LIN {X 0,Y 367.109,Z 392.803,A -85,B 0,C 180,E1 -12833.598,E2 -12833.598} C_VEL
LIN {X 0,Y 367.142,Z 392.339,A -85,B 0,C 180,E1 -12835.398,E2 -12835.398} C_VEL
LIN {X 0,Y 367.242,Z 390.593,A -85,B 0,C 180,E1 -12837.355,E2 -12837.355} C_VEL
LIN {X 0,Y 367.556,Z 387.382,A -85,B 0,C 180,E1 -12839.365,E2 -12839.365} C_VEL
LIN {X 0,Y 367.902,Z 382.367,A -85,B 0,C 180,E1 -12841.489,E2 -12841.489} C_VEL
LIN {X 0,Y 368.375,Z 376.663,A -85,B 0,C 180,E1 -12843.259,E2 -12843.259} C_VEL
LIN {X 0,Y 368.98,Z 369.858,A -85,B 0,C 180,E1 -12844.927,E2 -12844.927} C_VEL
LIN {X 0,Y 369.688,Z 362.048,A -85,B 0,C 180,E1 -12846.472,E2 -12846.472} C_VEL
LIN {X 0,Y 370.635,Z 352.269,A -85,B 0,C 180,E1 -12848.024,E2 -12848.024} C_VEL
LIN {X 0,Y 371.602,Z 341.593,A -85,B 0,C 180,E1 -12849.377,E2 -12849.377} C_VEL
LIN {X 0,Y 372.49,Z 331.477,A -85,B 0,C 180,E1 -12850.406,E2 -12850.406} C_VEL
LIN {X 0,Y 373.295,Z 320.016,A -85,B 0,C 180,E1 -12851.335,E2 -12851.335} C_VEL
LIN {X 0,Y 373.997,Z 307.877,A -85,B 0,C 180,E1 -12852.08,E2 -12852.08} C_VEL
LIN {X 0,Y 374.667,Z 294.33,A -85,B 0,C 180,E1 -12852.665,E2 -12852.665} C_VEL
LIN {X 0,Y 375.041,Z 279.803,A -85,B 0,C 180,E1 -12853.034,E2 -12853.034} C_VEL
LIN {X 0,Y 376.225,Z 207.722,A -85,B 0,C 180,E1 -12854.477,E2 -12854.477} C_VEL
LIN {X 0,Y 371.538,Z 182.162,A -85,B 0,C 180,E1 -12855.285,E2 -12855.285} C_VEL
LIN {X 0,Y 371.499,Z 181.295,A -85,B 0,C 180,E1 -12855.398,E2 -12855.398} C_VEL
LIN {X 0,Y 371.537,Z 177.576,A -85,B 0,C 180,E1 -12856.324,E2 -12856.324} C_VEL
LIN {X 0,Y 369.73,Z 167.61,A -85,B 0,C 180,E1 -12859.044,E2 -12859.044} C_VEL
LIN {X 0,Y 369.072,Z 164.061,A -85,B 0,C 180,E1 -12860.099,E2 -12860.099} C_VEL
LIN {X 0,Y 369.199,Z 163.994,A -85,B 0,C 180,E1 -12863.443,E2 -12863.443} C_VEL
LIN {X 0,Y 369.313,Z 163.984,A -85,B 0,C 180,E1 -12867.82,E2 -12867.82} C_VEL
LIN {X 0,Y 369.454,Z 163.964,A -85,B 0,C 180,E1 -12870.001,E2 -12870.001} C_VEL
LIN {X 0,Y 369.314,Z 163.98,A -85,B 0,C 180,E1 -12872.182,E2 -12872.182} C_VEL
LIN {X 0,Y 369.049,Z 164.011,A -85,B 0,C 180,E1 -12873.745,E2 -12873.745} C_VEL
LIN {X 0,Y 368.326,Z 164.102,A -85,B 0,C 180,E1 -12874.657,E2 -12874.657} C_VEL
LIN {X 0,Y 365.524,Z 164.452,A -85,B 0,C 180,E1 -12876.141,E2 -12876.141} C_VEL
LIN {X 0,Y 363.181,Z 164.746,A -85,B 0,C 180,E1 -12877.342,E2 -12877.342} C_VEL
LIN {X 0,Y 362.157,Z 164.871,A -85,B 0,C 180,E1 -12878.269,E2 -12878.269} C_VEL
LIN {X 0,Y 362.061,Z 164.882,A -85,B 0,C 180,E1 -12878.583,E2 -12878.583} C_VEL
LIN {X 0,Y 361.959,Z 164.894,A -85,B 0,C 180,E1 -12882.333,E2 -12882.333} C_VEL
LIN {X 0,Y 361.961,Z 164.894,A -85,B 0,C 180,E1 -12884.621,E2 -12884.621} C_VEL
LIN {X 0,Y 361.955,Z 164.895,A -85,B 0,C 180,E1 -12888.1,E2 -12888.1} C_VEL
LIN {X 0,Y 361.891,Z 164.905,A -85,B 0,C 180,E1 -12891.654,E2 -12891.654} C_VEL
LIN {X 0,Y 361.927,Z 164.904,A -85,B 0,C 180,E1 -12895.291,E2 -12895.291} C_VEL
LIN {X 0,Y 361.908,Z 164.902,A -85,B 0,C 180,E1 -12897.78,E2 -12897.78} C_VEL
LIN {X 0,Y 361.837,Z 164.911,A -85,B 0,C 180,E1 -12901.63,E2 -12901.63} C_VEL
LIN {X 0,Y 361.874,Z 164.908,A -85,B 0,C 180,E1 -12905.346,E2 -12905.346} C_VEL
LIN {X 0,Y 361.868,Z 164.911,A -85,B 0,C 180,E1 -12909.027,E2 -12909.027} C_VEL
LIN {X 0,Y 361.836,Z 164.916,A -85,B 0,C 180,E1 -12912.83,E2 -12912.83} C_VEL
LIN {X 0,Y 361.819,Z 164.912,A -85,B 0,C 180,E1 -12915.947,E2 -12915.947} C_VEL
LIN {X 0,Y 361.83,Z 164.912,A -85,B 0,C 180,E1 -12919.246,E2 -12919.246} C_VEL
LIN {X 0,Y 361.864,Z 164.909,A -85,B 0,C 180,E1 -12922.982,E2 -12922.982} C_VEL
LIN {X 0,Y 361.859,Z 164.912,A -85,B 0,C 180,E1 -12926.631,E2 -12926.631} C_VEL
LIN {X 0,Y 361.857,Z 164.907,A -85,B 0,C 180,E1 -12929.671,E2 -12929.671} C_VEL
LIN {X 0,Y 361.873,Z 164.905,A -85,B 0,C 180,E1 -12933.469,E2 -12933.469} C_VEL
LIN {X 0,Y 361.883,Z 164.904,A -85,B 0,C 180,E1 -12937.145,E2 -12937.145} C_VEL
LIN {X 0,Y 361.907,Z 164.902,A -85,B 0,C 180,E1 -12940.724,E2 -12940.724} C_VEL
LIN {X 0,Y 361.933,Z 164.898,A -85,B 0,C 180,E1 -12943.067,E2 -12943.067} C_VEL
LIN {X 0,Y 362,Z 164.891,A -85,B 0,C 180,E1 -12946.528,E2 -12946.528} C_VEL
LIN {X 0,Y 362,Z 164.895,A -85,B 0,C 180,E1 -12949.938,E2 -12949.938} C_VEL
LIN {X 0,Y 362.122,Z 164.875,A -85,B 0,C 180,E1 -12953.313,E2 -12953.313} C_VEL
LIN {X 0,Y 362.265,Z 164.862,A -85,B 0,C 180,E1 -12957.777,E2 -12957.777} C_VEL
LIN {X 0,Y 362.269,Z 164.857,A -85,B 0,C 180,E1 -12962.224,E2 -12962.224} C_VEL
LIN {X 0,Y 362.117,Z 164.875,A -85,B 0,C 180,E1 -12966.688,E2 -12966.688} C_VEL
LIN {X 0,Y 361.999,Z 164.891,A -85,B 0,C 180,E1 -12970.063,E2 -12970.063} C_VEL
LIN {X 0,Y 362.001,Z 164.891,A -85,B 0,C 180,E1 -12973.899,E2 -12973.899} C_VEL
LIN {X 0,Y 361.929,Z 164.9,A -85,B 0,C 180,E1 -12976.935,E2 -12976.935} C_VEL
LIN {X 0,Y 361.878,Z 164.904,A -85,B 0,C 180,E1 -12980.462,E2 -12980.462} C_VEL
LIN {X 0,Y 361.864,Z 164.906,A -85,B 0,C 180,E1 -12984.101,E2 -12984.101} C_VEL
LIN {X 0,Y 361.836,Z 164.911,A -85,B 0,C 180,E1 -12987.786,E2 -12987.786} C_VEL
LIN {X 0,Y 361.829,Z 164.915,A -85,B 0,C 180,E1 -12991.28,E2 -12991.28} C_VEL
LIN {X 0,Y 361.853,Z 164.908,A -85,B 0,C 180,E1 -12994.281,E2 -12994.281} C_VEL
LIN {X 0,Y 361.859,Z 164.91,A -85,B 0,C 180,E1 -12997.221,E2 -12997.221} C_VEL
LIN {X 0,Y 361.813,Z 164.917,A -85,B 0,C 180,E1 -13000.751,E2 -13000.751} C_VEL
LIN {X 0,Y 361.814,Z 164.914,A -85,B 0,C 180,E1 -13004.37,E2 -13004.37} C_VEL
LIN {X 0,Y 361.825,Z 164.911,A -85,B 0,C 180,E1 -13007.571,E2 -13007.571} C_VEL
LIN {X 0,Y 361.842,Z 164.909,A -85,B 0,C 180,E1 -13011.571,E2 -13011.571} C_VEL
LIN {X 0,Y 361.865,Z 164.912,A -85,B 0,C 180,E1 -13014.658,E2 -13014.658} C_VEL
LIN {X 0,Y 361.822,Z 164.916,A -85,B 0,C 180,E1 -13018.368,E2 -13018.368} C_VEL
LIN {X 0,Y 361.909,Z 165.145,A -85,B 0,C 180,E1 -13021.392,E2 -13021.392} C_VEL
LIN {X 0,Y 364.539,Z 178.239,A -85,B 0,C 180,E1 -13024.903,E2 -13024.903} C_VEL
LIN {X 0,Y 365.265,Z 183.174,A -85,B 0,C 180,E1 -13026.167,E2 -13026.167} C_VEL
LIN {X 0,Y 364.446,Z 192.349,A -85,B 0,C 180,E1 -13028.323,E2 -13028.323} C_VEL
LIN {X 0,Y 365.484,Z 198.9,A -85,B 0,C 180,E1 -13028.57,E2 -13028.57} C_VEL
LIN {X 0,Y 369.443,Z 223.822,A -85,B 0,C 180,E1 -13029.318,E2 -13029.318} C_VEL
LIN {X 0,Y 367.995,Z 300.62,A -85,B 0,C 180,E1 -13030.909,E2 -13030.909} C_VEL
LIN {X 0,Y 367.351,Z 314.312,A -85,B 0,C 180,E1 -13031.417,E2 -13031.417} C_VEL
LIN {X 0,Y 366.485,Z 327.23,A -85,B 0,C 180,E1 -13032.131,E2 -13032.131} C_VEL
LIN {X 0,Y 365.522,Z 339.819,A -85,B 0,C 180,E1 -13033.092,E2 -13033.092} C_VEL
LIN {X 0,Y 364.556,Z 351.066,A -85,B 0,C 180,E1 -13034.198,E2 -13034.198} C_VEL
LIN {X 0,Y 363.668,Z 361.183,A -85,B 0,C 180,E1 -13035.449,E2 -13035.449} C_VEL
LIN {X 0,Y 362.79,Z 370.328,A -85,B 0,C 180,E1 -13036.842,E2 -13036.842} C_VEL
LIN {X 0,Y 361.84,Z 379.24,A -85,B 0,C 180,E1 -13038.516,E2 -13038.516} C_VEL
LIN {X 0,Y 361.199,Z 386.366,A -85,B 0,C 180,E1 -13040.196,E2 -13040.196} C_VEL
LIN {X 0,Y 360.687,Z 392.862,A -85,B 0,C 180,E1 -13042.16,E2 -13042.16} C_VEL
LIN {X 0,Y 360.428,Z 397.403,A -85,B 0,C 180,E1 -13043.965,E2 -13043.965} C_VEL
LIN {X 0,Y 360.348,Z 400.313,A -85,B 0,C 180,E1 -13045.525,E2 -13045.525} C_VEL
LIN {X 0,Y 360.275,Z 401.892,A -85,B 0,C 180,E1 -13046.644,E2 -13046.644} C_VEL
LIN {X 0,Y 360.226,Z 403.034,A -85,B 0,C 180,E1 -13047.763,E2 -13047.763} C_VEL
LIN {X 0,Y 360.252,Z 403.744,A -85,B 0,C 180,E1 -13048.881,E2 -13048.881} C_VEL
LIN {X 0,Y 360.291,Z 404.061,A -85,B 0,C 180,E1 -13049.999,E2 -13049.999} C_VEL
LIN {X 0,Y 360.25,Z 403.987,A -85,B 0,C 180,E1 -13051.117,E2 -13051.117} C_VEL
LIN {X 0,Y 360.225,Z 403.495,A -85,B 0,C 180,E1 -13052.235,E2 -13052.235} C_VEL
LIN {X 0,Y 360.278,Z 402.578,A -85,B 0,C 180,E1 -13053.354,E2 -13053.354} C_VEL
LIN {X 0,Y 360.379,Z 401.262,A -85,B 0,C 180,E1 -13054.473,E2 -13054.473} C_VEL
LIN {X 0,Y 360.463,Z 398.611,A -85,B 0,C 180,E1 -13056.087,E2 -13056.087} C_VEL
LIN {X 0,Y 360.756,Z 394.67,A -85,B 0,C 180,E1 -13057.836,E2 -13057.836} C_VEL
LIN {X 0,Y 361.219,Z 389.732,A -85,B 0,C 180,E1 -13059.518,E2 -13059.518} C_VEL
LIN {X 0,Y 361.871,Z 383.528,A -85,B 0,C 180,E1 -13061.197,E2 -13061.197} C_VEL
LIN {X 0,Y 362.818,Z 375.82,A -85,B 0,C 180,E1 -13062.87,E2 -13062.87} C_VEL
LIN {X 0,Y 364.016,Z 366.15,A -85,B 0,C 180,E1 -13064.535,E2 -13064.535} C_VEL
LIN {X 0,Y 365.018,Z 356.196,A -85,B 0,C 180,E1 -13065.923,E2 -13065.923} C_VEL
LIN {X 0,Y 366.289,Z 344.984,A -85,B 0,C 180,E1 -13067.156,E2 -13067.156} C_VEL
LIN {X 0,Y 367.386,Z 334.036,A -85,B 0,C 180,E1 -13068.109,E2 -13068.109} C_VEL
LIN {X 0,Y 368.435,Z 321.974,A -85,B 0,C 180,E1 -13068.92,E2 -13068.92} C_VEL
LIN {X 0,Y 369.204,Z 309.573,A -85,B 0,C 180,E1 -13069.529,E2 -13069.529} C_VEL
LIN {X 0,Y 369.741,Z 295.528,A -85,B 0,C 180,E1 -13069.97,E2 -13069.97} C_VEL
LIN {X 0,Y 371.27,Z 223.76,A -85,B 0,C 180,E1 -13071.458,E2 -13071.458} C_VEL
LIN {X 0,Y 367.556,Z 202.377,A -85,B 0,C 180,E1 -13072.204,E2 -13072.204} C_VEL
LIN {X 0,Y 365.353,Z 191.898,A -85,B 0,C 180,E1 -13072.644,E2 -13072.644} C_VEL
LIN {X 0,Y 365.684,Z 187.966,A -85,B 0,C 180,E1 -13073.501,E2 -13073.501} C_VEL
LIN {X 0,Y 365.843,Z 184.32,A -85,B 0,C 180,E1 -13074.393,E2 -13074.393} C_VEL
LIN {X 0,Y 364.208,Z 175.338,A -85,B 0,C 180,E1 -13076.802,E2 -13076.802} C_VEL
LIN {X 0,Y 361.879,Z 164.958,A -85,B 0,C 180,E1 -13079.803,E2 -13079.803} C_VEL
LIN {X 0,Y 361.853,Z 164.907,A -85,B 0,C 180,E1 -13083.367,E2 -13083.367} C_VEL
LIN {X 0,Y 361.855,Z 164.911,A -85,B 0,C 180,E1 -13087.017,E2 -13087.017} C_VEL
LIN {X 0,Y 361.804,Z 164.917,A -85,B 0,C 180,E1 -13090.749,E2 -13090.749} C_VEL
LIN {X 0,Y 361.804,Z 164.914,A -85,B 0,C 180,E1 -13094.368,E2 -13094.368} C_VEL
LIN {X 0,Y 361.814,Z 164.918,A -85,B 0,C 180,E1 -13097.569,E2 -13097.569} C_VEL
LIN {X 0,Y 361.834,Z 164.91,A -85,B 0,C 180,E1 -13101.57,E2 -13101.57} C_VEL
LIN {X 0,Y 361.861,Z 164.91,A -85,B 0,C 180,E1 -13104.655,E2 -13104.655} C_VEL
LIN {X 0,Y 361.828,Z 164.912,A -85,B 0,C 180,E1 -13108.369,E2 -13108.369} C_VEL
LIN {X 0,Y 361.856,Z 164.913,A -85,B 0,C 180,E1 -13110.951,E2 -13110.951} C_VEL
LIN {X 0,Y 361.869,Z 164.91,A -85,B 0,C 180,E1 -13114.705,E2 -13114.705} C_VEL
LIN {X 0,Y 361.849,Z 164.909,A -85,B 0,C 180,E1 -13118.344,E2 -13118.344} C_VEL
LIN {X 0,Y 361.909,Z 164.9,A -85,B 0,C 180,E1 -13122.084,E2 -13122.084} C_VEL
LIN {X 0,Y 361.95,Z 164.894,A -85,B 0,C 180,E1 -13125.379,E2 -13125.379} C_VEL
LIN {X 0,Y 361.957,Z 164.892,A -85,B 0,C 180,E1 -13128.803,E2 -13128.803} C_VEL
LIN {X 0,Y 362.082,Z 164.879,A -85,B 0,C 180,E1 -13132.191,E2 -13132.191} C_VEL
LIN {X 0,Y 362.089,Z 164.881,A -85,B 0,C 180,E1 -13134.43,E2 -13134.43} C_VEL
LIN {X 0,Y 362.255,Z 164.858,A -85,B 0,C 180,E1 -13137.776,E2 -13137.776} C_VEL
LIN {X 0,Y 362.252,Z 164.863,A -85,B 0,C 180,E1 -13142.223,E2 -13142.223} C_VEL
LIN {X 0,Y 362.127,Z 164.875,A -85,B 0,C 180,E1 -13146.686,E2 -13146.686} C_VEL
LIN {X 0,Y 361.982,Z 164.894,A -85,B 0,C 180,E1 -13150.063,E2 -13150.063} C_VEL
LIN {X 0,Y 361.985,Z 164.893,A -85,B 0,C 180,E1 -13153.898,E2 -13153.898} C_VEL
LIN {X 0,Y 361.915,Z 164.904,A -85,B 0,C 180,E1 -13156.934,E2 -13156.934} C_VEL
LIN {X 0,Y 361.87,Z 164.91,A -85,B 0,C 180,E1 -13160.461,E2 -13160.461} C_VEL
LIN {X 0,Y 361.848,Z 164.915,A -85,B 0,C 180,E1 -13164.101,E2 -13164.101} C_VEL
LIN {X 0,Y 361.861,Z 165.115,A -85,B 0,C 180,E1 -13166.7,E2 -13166.7} C_VEL
LIN {X 0,Y 364.298,Z 175.702,A -85,B 0,C 180,E1 -13169.761,E2 -13169.761} C_VEL
LIN {X 0,Y 365.43,Z 181.869,A -85,B 0,C 180,E1 -13171.387,E2 -13171.387} C_VEL
LIN {X 0,Y 366.56,Z 185.876,A -85,B 0,C 180,E1 -13171.619,E2 -13171.619} C_VEL
LIN {X 0,Y 370.397,Z 203.475,A -85,B 0,C 180,E1 -13172.3,E2 -13172.3} C_VEL
LIN {X 0,Y 371.577,Z 210.184,A -85,B 0,C 180,E1 -13172.534,E2 -13172.534} C_VEL
LIN {X 0,Y 369.736,Z 290.324,A -85,B 0,C 180,E1 -13174.219,E2 -13174.219} C_VEL
LIN {X 0,Y 369.122,Z 303.569,A -85,B 0,C 180,E1 -13174.721,E2 -13174.721} C_VEL
LIN {X 0,Y 368.374,Z 315.12,A -85,B 0,C 180,E1 -13175.357,E2 -13175.357} C_VEL
LIN {X 0,Y 367.382,Z 327.182,A -85,B 0,C 180,E1 -13176.248,E2 -13176.248} C_VEL
LIN {X 0,Y 366.166,Z 339.44,A -85,B 0,C 180,E1 -13177.431,E2 -13177.431} C_VEL
LIN {X 0,Y 364.915,Z 350.146,A -85,B 0,C 180,E1 -13178.742,E2 -13178.742} C_VEL
LIN {X 0,Y 363.768,Z 359.977,A -85,B 0,C 180,E1 -13180.261,E2 -13180.261} C_VEL
LIN {X 0,Y 362.806,Z 367.927,A -85,B 0,C 180,E1 -13181.776,E2 -13181.776} C_VEL
LIN {X 0,Y 361.922,Z 374.835,A -85,B 0,C 180,E1 -13183.394,E2 -13183.394} C_VEL
LIN {X 0,Y 361.379,Z 380.255,A -85,B 0,C 180,E1 -13184.978,E2 -13184.978} C_VEL
LIN {X 0,Y 360.798,Z 385.639,A -85,B 0,C 180,E1 -13187.021,E2 -13187.021} C_VEL
LIN {X 0,Y 360.557,Z 388.562,A -85,B 0,C 180,E1 -13188.494,E2 -13188.494} C_VEL
LIN {X 0,Y 360.302,Z 390.657,A -85,B 0,C 180,E1 -13189.935,E2 -13189.935} C_VEL
LIN {X 0,Y 360.123,Z 392.042,A -85,B 0,C 180,E1 -13191.357,E2 -13191.357} C_VEL
LIN {X 0,Y 360.005,Z 392.863,A -85,B 0,C 180,E1 -13193.167,E2 -13193.167} C_VEL
LIN {X 0,Y 360.039,Z 392.591,A -85,B 0,C 180,E1 -13195.068,E2 -13195.068} C_VEL
LIN {X 0,Y 360.11,Z 391.067,A -85,B 0,C 180,E1 -13197.055,E2 -13197.055} C_VEL
LIN {X 0,Y 360.416,Z 388.143,A -85,B 0,C 180,E1 -13199.09,E2 -13199.09} C_VEL
LIN {X 0,Y 360.663,Z 384.41,A -85,B 0,C 180,E1 -13200.848,E2 -13200.848} C_VEL
LIN {X 0,Y 361.144,Z 378.85,A -85,B 0,C 180,E1 -13202.788,E2 -13202.788} C_VEL
LIN {X 0,Y 361.771,Z 371.726,A -85,B 0,C 180,E1 -13204.7,E2 -13204.7} C_VEL
LIN {X 0,Y 362.471,Z 364.27,A -85,B 0,C 180,E1 -13206.278,E2 -13206.278} C_VEL
LIN {X 0,Y 363.303,Z 355.984,A -85,B 0,C 180,E1 -13207.709,E2 -13207.709} C_VEL
LIN {X 0,Y 364.275,Z 346.17,A -85,B 0,C 180,E1 -13209.09,E2 -13209.09} C_VEL
LIN {X 0,Y 365.334,Z 334.976,A -85,B 0,C 180,E1 -13210.35,E2 -13210.35} C_VEL
LIN {X 0,Y 366.278,Z 323.048,A -85,B 0,C 180,E1 -13211.399,E2 -13211.399} C_VEL
LIN {X 0,Y 367.069,Z 310.254,A -85,B 0,C 180,E1 -13212.259,E2 -13212.259} C_VEL
LIN {X 0,Y 367.727,Z 297.524,A -85,B 0,C 180,E1 -13212.86,E2 -13212.86} C_VEL
LIN {X 0,Y 368.207,Z 283.92,A -85,B 0,C 180,E1 -13213.268,E2 -13213.268} C_VEL
LIN {X 0,Y 369.42,Z 208.091,A -85,B 0,C 180,E1 -13214.823,E2 -13214.823} C_VEL
LIN {X 0,Y 364.629,Z 182.094,A -85,B 0,C 180,E1 -13215.669,E2 -13215.669} C_VEL
LIN {X 0,Y 364.61,Z 179.145,A -85,B 0,C 180,E1 -13216.344,E2 -13216.344} C_VEL
LIN {X 0,Y 363.008,Z 170.131,A -85,B 0,C 180,E1 -13218.838,E2 -13218.838} C_VEL
LIN {X 0,Y 362.031,Z 164.963,A -85,B 0,C 180,E1 -13220.363,E2 -13220.363} C_VEL
LIN {X 0,Y 362.161,Z 164.87,A -85,B 0,C 180,E1 -13223.315,E2 -13223.315} C_VEL
LIN {X 0,Y 362.277,Z 164.861,A -85,B 0,C 180,E1 -13227.778,E2 -13227.778} C_VEL
LIN {X 0,Y 362.424,Z 164.84,A -85,B 0,C 180,E1 -13230.001,E2 -13230.001} C_VEL
LIN {X 0,Y 362.278,Z 164.856,A -85,B 0,C 180,E1 -13232.225,E2 -13232.225} C_VEL
LIN {X 0,Y 362.147,Z 164.871,A -85,B 0,C 180,E1 -13236.688,E2 -13236.688} C_VEL
LIN {X 0,Y 362.061,Z 164.882,A -85,B 0,C 180,E1 -13238.583,E2 -13238.583} C_VEL
LIN {X 0,Y 361.343,Z 164.977,A -85,B 0,C 180,E1 -13239.51,E2 -13239.51} C_VEL
LIN {X 0,Y 358.425,Z 165.336,A -85,B 0,C 180,E1 -13241.018,E2 -13241.018} C_VEL
LIN {X 0,Y 356,Z 165.637,A -85,B 0,C 180,E1 -13242.238,E2 -13242.238} C_VEL
LIN {X 0,Y 354.995,Z 165.765,A -85,B 0,C 180,E1 -13243.183,E2 -13243.183} C_VEL
LIN {X 0,Y 354.932,Z 165.771,A -85,B 0,C 180,E1 -13243.502,E2 -13243.502} C_VEL
LIN {X 0,Y 354.897,Z 165.779,A -85,B 0,C 180,E1 -13247.281,E2 -13247.281} C_VEL
LIN {X 0,Y 354.839,Z 165.784,A -85,B 0,C 180,E1 -13250.887,E2 -13250.887} C_VEL
LIN {X 0,Y 354.861,Z 165.779,A -85,B 0,C 180,E1 -13254.577,E2 -13254.577} C_VEL
LIN {X 0,Y 354.881,Z 165.782,A -85,B 0,C 180,E1 -13257.097,E2 -13257.097} C_VEL
LIN {X 0,Y 354.799,Z 165.792,A -85,B 0,C 180,E1 -13260.999,E2 -13260.999} C_VEL
LIN {X 0,Y 354.806,Z 165.786,A -85,B 0,C 180,E1 -13263.703,E2 -13263.703} C_VEL
LIN {X 0,Y 354.797,Z 165.788,A -85,B 0,C 180,E1 -13266.46,E2 -13266.46} C_VEL
LIN {X 0,Y 354.824,Z 165.785,A -85,B 0,C 180,E1 -13269.424,E2 -13269.424} C_VEL
LIN {X 0,Y 354.788,Z 165.793,A -85,B 0,C 180,E1 -13272.868,E2 -13272.868} C_VEL
LIN {X 0,Y 354.768,Z 165.791,A -85,B 0,C 180,E1 -13276.104,E2 -13276.104} C_VEL
LIN {X 0,Y 354.782,Z 165.79,A -85,B 0,C 180,E1 -13279.179,E2 -13279.179} C_VEL
LIN {X 0,Y 354.801,Z 165.79,A -85,B 0,C 180,E1 -13282.405,E2 -13282.405} C_VEL
LIN {X 0,Y 354.812,Z 165.787,A -85,B 0,C 180,E1 -13284.941,E2 -13284.941} C_VEL
LIN {X 0,Y 354.794,Z 165.792,A -85,B 0,C 180,E1 -13288.406,E2 -13288.406} C_VEL
LIN {X 0,Y 354.802,Z 165.786,A -85,B 0,C 180,E1 -13291.615,E2 -13291.615} C_VEL
LIN {X 0,Y 354.852,Z 165.78,A -85,B 0,C 180,E1 -13295.424,E2 -13295.424} C_VEL
LIN {X 0,Y 354.828,Z 165.783,A -85,B 0,C 180,E1 -13299.114,E2 -13299.114} C_VEL
LIN {X 0,Y 354.9,Z 165.775,A -85,B 0,C 180,E1 -13302.721,E2 -13302.721} C_VEL
LIN {X 0,Y 354.953,Z 165.772,A -85,B 0,C 180,E1 -13306.256,E2 -13306.256} C_VEL
LIN {X 0,Y 354.956,Z 165.77,A -85,B 0,C 180,E1 -13309.736,E2 -13309.736} C_VEL
LIN {X 0,Y 355.088,Z 165.751,A -85,B 0,C 180,E1 -13313.18,E2 -13313.18} C_VEL
LIN {X 0,Y 355.227,Z 165.738,A -85,B 0,C 180,E1 -13317.733,E2 -13317.733} C_VEL
LIN {X 0,Y 355.146,Z 165.744,A -85,B 0,C 180,E1 -13321.134,E2 -13321.134} C_VEL
LIN {X 0,Y 355.232,Z 165.734,A -85,B 0,C 180,E1 -13322.268,E2 -13322.268} C_VEL
LIN {X 0,Y 355.084,Z 165.751,A -85,B 0,C 180,E1 -13326.821,E2 -13326.821} C_VEL
LIN {X 0,Y 354.955,Z 165.767,A -85,B 0,C 180,E1 -13330.265,E2 -13330.265} C_VEL
LIN {X 0,Y 354.945,Z 165.769,A -85,B 0,C 180,E1 -13334.019,E2 -13334.019} C_VEL
LIN {X 0,Y 354.881,Z 165.781,A -85,B 0,C 180,E1 -13337.281,E2 -13337.281} C_VEL
LIN {X 0,Y 354.82,Z 165.789,A -85,B 0,C 180,E1 -13341.417,E2 -13341.417} C_VEL
LIN {X 0,Y 354.806,Z 165.786,A -85,B 0,C 180,E1 -13344.581,E2 -13344.581} C_VEL
LIN {X 0,Y 354.791,Z 165.788,A -85,B 0,C 180,E1 -13348.387,E2 -13348.387} C_VEL
LIN {X 0,Y 354.782,Z 165.789,A -85,B 0,C 180,E1 -13352.334,E2 -13352.334} C_VEL
LIN {X 0,Y 354.821,Z 165.784,A -85,B 0,C 180,E1 -13355.698,E2 -13355.698} C_VEL
LIN {X 0,Y 354.772,Z 165.791,A -85,B 0,C 180,E1 -13359.412,E2 -13359.412} C_VEL
LIN {X 0,Y 354.784,Z 165.794,A -85,B 0,C 180,E1 -13362.866,E2 -13362.866} C_VEL
LIN {X 0,Y 354.765,Z 165.791,A -85,B 0,C 180,E1 -13366.103,E2 -13366.103} C_VEL
LIN {X 0,Y 354.766,Z 165.792,A -85,B 0,C 180,E1 -13369.175,E2 -13369.175} C_VEL
LIN {X 0,Y 354.799,Z 165.79,A -85,B 0,C 180,E1 -13372.405,E2 -13372.405} C_VEL
LIN {X 0,Y 354.802,Z 165.789,A -85,B 0,C 180,E1 -13374.939,E2 -13374.939} C_VEL
LIN {X 0,Y 354.777,Z 165.794,A -85,B 0,C 180,E1 -13378.41,E2 -13378.41} C_VEL
LIN {X 0,Y 354.827,Z 165.885,A -85,B 0,C 180,E1 -13381.013,E2 -13381.013} C_VEL
LIN {X 0,Y 357.28,Z 177.904,A -85,B 0,C 180,E1 -13384.356,E2 -13384.356} C_VEL
LIN {X 0,Y 358.289,Z 184.081,A -85,B 0,C 180,E1 -13385.981,E2 -13385.981} C_VEL
LIN {X 0,Y 357.549,Z 192.4,A -85,B 0,C 180,E1 -13387.954,E2 -13387.954} C_VEL
LIN {X 0,Y 362.726,Z 224.91,A -85,B 0,C 180,E1 -13388.988,E2 -13388.988} C_VEL
LIN {X 0,Y 361.247,Z 300.218,A -85,B 0,C 180,E1 -13390.575,E2 -13390.575} C_VEL
LIN {X 0,Y 360.572,Z 313.996,A -85,B 0,C 180,E1 -13391.092,E2 -13391.092} C_VEL
LIN {X 0,Y 359.743,Z 326.459,A -85,B 0,C 180,E1 -13391.784,E2 -13391.784} C_VEL
LIN {X 0,Y 358.855,Z 337.615,A -85,B 0,C 180,E1 -13392.622,E2 -13392.622} C_VEL
LIN {X 0,Y 357.766,Z 349.237,A -85,B 0,C 180,E1 -13393.743,E2 -13393.743} C_VEL
LIN {X 0,Y 356.937,Z 359.032,A -85,B 0,C 180,E1 -13394.929,E2 -13394.929} C_VEL
LIN {X 0,Y 355.994,Z 368.286,A -85,B 0,C 180,E1 -13396.295,E2 -13396.295} C_VEL
LIN {X 0,Y 354.97,Z 377.546,A -85,B 0,C 180,E1 -13398,E2 -13398} C_VEL
LIN {X 0,Y 354.272,Z 384.99,A -85,B 0,C 180,E1 -13399.714,E2 -13399.714} C_VEL
LIN {X 0,Y 353.778,Z 390.952,A -85,B 0,C 180,E1 -13401.43,E2 -13401.43} C_VEL
LIN {X 0,Y 353.42,Z 395.641,A -85,B 0,C 180,E1 -13403.146,E2 -13403.146} C_VEL
LIN {X 0,Y 353.25,Z 399.198,A -85,B 0,C 180,E1 -13404.862,E2 -13404.862} C_VEL
LIN {X 0,Y 353.199,Z 401.729,A -85,B 0,C 180,E1 -13406.577,E2 -13406.577} C_VEL
LIN {X 0,Y 353.136,Z 402.894,A -85,B 0,C 180,E1 -13407.718,E2 -13407.718} C_VEL
LIN {X 0,Y 353.151,Z 403.616,A -85,B 0,C 180,E1 -13408.859,E2 -13408.859} C_VEL
LIN {X 0,Y 353.192,Z 403.945,A -85,B 0,C 180,E1 -13409.999,E2 -13409.999} C_VEL
LIN {X 0,Y 353.15,Z 403.881,A -85,B 0,C 180,E1 -13411.139,E2 -13411.139} C_VEL
LIN {X 0,Y 353.136,Z 403.41,A -85,B 0,C 180,E1 -13412.28,E2 -13412.28} C_VEL
LIN {X 0,Y 353.203,Z 402.503,A -85,B 0,C 180,E1 -13413.421,E2 -13413.421} C_VEL
LIN {X 0,Y 353.294,Z 401.2,A -85,B 0,C 180,E1 -13414.563,E2 -13414.563} C_VEL
LIN {X 0,Y 353.389,Z 398.822,A -85,B 0,C 180,E1 -13416.078,E2 -13416.078} C_VEL
LIN {X 0,Y 353.71,Z 394.663,A -85,B 0,C 180,E1 -13417.994,E2 -13417.994} C_VEL
LIN {X 0,Y 354.187,Z 389.761,A -85,B 0,C 180,E1 -13419.709,E2 -13419.709} C_VEL
LIN {X 0,Y 354.873,Z 383.591,A -85,B 0,C 180,E1 -13421.421,E2 -13421.421} C_VEL
LIN {X 0,Y 355.905,Z 375.927,A -85,B 0,C 180,E1 -13423.124,E2 -13423.124} C_VEL
LIN {X 0,Y 357.133,Z 366.308,A -85,B 0,C 180,E1 -13424.821,E2 -13424.821} C_VEL
LIN {X 0,Y 358.202,Z 356.405,A -85,B 0,C 180,E1 -13426.234,E2 -13426.234} C_VEL
LIN {X 0,Y 359.536,Z 345.296,A -85,B 0,C 180,E1 -13427.489,E2 -13427.489} C_VEL
LIN {X 0,Y 360.487,Z 336.205,A -85,B 0,C 180,E1 -13428.321,E2 -13428.321} C_VEL
LIN {X 0,Y 361.626,Z 323.65,A -85,B 0,C 180,E1 -13429.217,E2 -13429.217} C_VEL
LIN {X 0,Y 362.533,Z 310.484,A -85,B 0,C 180,E1 -13429.904,E2 -13429.904} C_VEL
LIN {X 0,Y 363.187,Z 297.192,A -85,B 0,C 180,E1 -13430.346,E2 -13430.346} C_VEL
LIN {X 0,Y 364.776,Z 224.593,A -85,B 0,C 180,E1 -13431.895,E2 -13431.895} C_VEL
LIN {X 0,Y 360.877,Z 202.469,A -85,B 0,C 180,E1 -13432.694,E2 -13432.694} C_VEL
LIN {X 0,Y 358.624,Z 191.839,A -85,B 0,C 180,E1 -13433.15,E2 -13433.15} C_VEL
LIN {X 0,Y 358.815,Z 189.342,A -85,B 0,C 180,E1 -13433.672,E2 -13433.672} C_VEL
LIN {X 0,Y 358.97,Z 185.71,A -85,B 0,C 180,E1 -13434.583,E2 -13434.583} C_VEL
LIN {X 0,Y 357.417,Z 177.298,A -85,B 0,C 180,E1 -13436.887,E2 -13436.887} C_VEL
LIN {X 0,Y 354.863,Z 166.034,A -85,B 0,C 180,E1 -13440.167,E2 -13440.167} C_VEL
LIN {X 0,Y 354.773,Z 165.792,A -85,B 0,C 180,E1 -13441.589,E2 -13441.589} C_VEL
LIN {X 0,Y 354.803,Z 165.79,A -85,B 0,C 180,E1 -13445.058,E2 -13445.058} C_VEL
LIN {X 0,Y 354.787,Z 165.791,A -85,B 0,C 180,E1 -13447.883,E2 -13447.883} C_VEL
LIN {X 0,Y 354.761,Z 165.797,A -85,B 0,C 180,E1 -13451.166,E2 -13451.166} C_VEL
LIN {X 0,Y 354.75,Z 165.793,A -85,B 0,C 180,E1 -13454.503,E2 -13454.503} C_VEL
LIN {X 0,Y 354.774,Z 165.795,A -85,B 0,C 180,E1 -13457.659,E2 -13457.659} C_VEL
LIN {X 0,Y 354.777,Z 165.792,A -85,B 0,C 180,E1 -13460.66,E2 -13460.66} C_VEL
LIN {X 0,Y 354.809,Z 165.787,A -85,B 0,C 180,E1 -13464.3,E2 -13464.3} C_VEL
LIN {X 0,Y 354.777,Z 165.791,A -85,B 0,C 180,E1 -13467.665,E2 -13467.665} C_VEL
LIN {X 0,Y 354.787,Z 165.788,A -85,B 0,C 180,E1 -13471.613,E2 -13471.613} C_VEL
LIN {X 0,Y 354.824,Z 165.783,A -85,B 0,C 180,E1 -13475.656,E2 -13475.656} C_VEL
LIN {X 0,Y 354.814,Z 165.787,A -85,B 0,C 180,E1 -13479.112,E2 -13479.112} C_VEL
LIN {X 0,Y 354.868,Z 165.781,A -85,B 0,C 180,E1 -13482.718,E2 -13482.718} C_VEL
LIN {X 0,Y 354.94,Z 165.769,A -85,B 0,C 180,E1 -13486.254,E2 -13486.254} C_VEL
LIN {X 0,Y 354.943,Z 165.768,A -85,B 0,C 180,E1 -13489.734,E2 -13489.734} C_VEL
LIN {X 0,Y 355.093,Z 165.748,A -85,B 0,C 180,E1 -13493.179,E2 -13493.179} C_VEL
LIN {X 0,Y 355.218,Z 165.735,A -85,B 0,C 180,E1 -13497.732,E2 -13497.732} C_VEL
LIN {X 0,Y 355.214,Z 165.739,A -85,B 0,C 180,E1 -13502.267,E2 -13502.267} C_VEL
LIN {X 0,Y 355.092,Z 165.752,A -85,B 0,C 180,E1 -13506.82,E2 -13506.82} C_VEL
LIN {X 0,Y 354.938,Z 165.774,A -85,B 0,C 180,E1 -13510.265,E2 -13510.265} C_VEL
LIN {X 0,Y 354.929,Z 165.772,A -85,B 0,C 180,E1 -13514.018,E2 -13514.018} C_VEL
LIN {X 0,Y 354.877,Z 165.781,A -85,B 0,C 180,E1 -13518.092,E2 -13518.092} C_VEL
LIN {X 0,Y 354.801,Z 165.791,A -85,B 0,C 180,E1 -13522.108,E2 -13522.108} C_VEL
LIN {X 0,Y 354.809,Z 165.808,A -85,B 0,C 180,E1 -13526.071,E2 -13526.071} C_VEL
LIN {X 0,Y 354.963,Z 166.64,A -85,B 0,C 180,E1 -13526.454,E2 -13526.454} C_VEL
LIN {X 0,Y 357.347,Z 176.861,A -85,B 0,C 180,E1 -13529.45,E2 -13529.45} C_VEL
LIN {X 0,Y 358.375,Z 182.138,A -85,B 0,C 180,E1 -13530.859,E2 -13530.859} C_VEL
LIN {X 0,Y 360.347,Z 188.103,A -85,B 0,C 180,E1 -13531.202,E2 -13531.202} C_VEL
LIN {X 0,Y 364.167,Z 205.794,A -85,B 0,C 180,E1 -13531.901,E2 -13531.901} C_VEL
LIN {X 0,Y 365.065,Z 212.031,A -85,B 0,C 180,E1 -13532.11,E2 -13532.11} C_VEL
LIN {X 0,Y 363.179,Z 290.114,A -85,B 0,C 180,E1 -13533.787,E2 -13533.787} C_VEL
LIN {X 0,Y 362.539,Z 303.278,A -85,B 0,C 180,E1 -13534.29,E2 -13534.29} C_VEL
LIN {X 0,Y 361.75,Z 315.235,A -85,B 0,C 180,E1 -13534.958,E2 -13534.958} C_VEL
LIN {X 0,Y 360.71,Z 327.291,A -85,B 0,C 180,E1 -13535.863,E2 -13535.863} C_VEL
LIN {X 0,Y 359.544,Z 338.417,A -85,B 0,C 180,E1 -13536.942,E2 -13536.942} C_VEL
LIN {X 0,Y 358.426,Z 347.741,A -85,B 0,C 180,E1 -13538.06,E2 -13538.06} C_VEL
LIN {X 0,Y 357.311,Z 356.91,A -85,B 0,C 180,E1 -13539.406,E2 -13539.406} C_VEL
LIN {X 0,Y 356.201,Z 365.669,A -85,B 0,C 180,E1 -13540.99,E2 -13540.99} C_VEL
LIN {X 0,Y 355.289,Z 372.763,A -85,B 0,C 180,E1 -13542.58,E2 -13542.58} C_VEL
LIN {X 0,Y 354.445,Z 379.441,A -85,B 0,C 180,E1 -13544.456,E2 -13544.456} C_VEL
LIN {X 0,Y 353.953,Z 383.735,A -85,B 0,C 180,E1 -13545.979,E2 -13545.979} C_VEL
LIN {X 0,Y 353.639,Z 387.135,A -85,B 0,C 180,E1 -13547.494,E2 -13547.494} C_VEL
LIN {X 0,Y 353.32,Z 389.861,A -85,B 0,C 180,E1 -13549.101,E2 -13549.101} C_VEL
LIN {X 0,Y 353.049,Z 391.916,A -85,B 0,C 180,E1 -13550.927,E2 -13550.927} C_VEL
LIN {X 0,Y 352.928,Z 392.933,A -85,B 0,C 180,E1 -13552.8,E2 -13552.8} C_VEL
LIN {X 0,Y 352.934,Z 392.841,A -85,B 0,C 180,E1 -13554.729,E2 -13554.729} C_VEL
LIN {X 0,Y 352.982,Z 391.51,A -85,B 0,C 180,E1 -13556.744,E2 -13556.744} C_VEL
LIN {X 0,Y 353.279,Z 388.743,A -85,B 0,C 180,E1 -13558.855,E2 -13558.855} C_VEL
LIN {X 0,Y 353.601,Z 384.405,A -85,B 0,C 180,E1 -13560.987,E2 -13560.987} C_VEL
LIN {X 0,Y 354.064,Z 379.22,A -85,B 0,C 180,E1 -13562.838,E2 -13562.838} C_VEL
LIN {X 0,Y 354.723,Z 372.155,A -85,B 0,C 180,E1 -13564.79,E2 -13564.79} C_VEL
LIN {X 0,Y 355.453,Z 364.784,A -85,B 0,C 180,E1 -13566.4,E2 -13566.4} C_VEL
LIN {X 0,Y 356.398,Z 355.693,A -85,B 0,C 180,E1 -13567.998,E2 -13567.998} C_VEL
LIN {X 0,Y 357.401,Z 345.738,A -85,B 0,C 180,E1 -13569.413,E2 -13569.413} C_VEL
LIN {X 0,Y 358.496,Z 334.499,A -85,B 0,C 180,E1 -13570.683,E2 -13570.683} C_VEL
LIN {X 0,Y 359.478,Z 322.167,A -85,B 0,C 180,E1 -13571.773,E2 -13571.773} C_VEL
LIN {X 0,Y 360.263,Z 310.462,A -85,B 0,C 180,E1 -13572.562,E2 -13572.562} C_VEL
LIN {X 0,Y 360.938,Z 297.555,A -85,B 0,C 180,E1 -13573.183,E2 -13573.183} C_VEL
LIN {X 0,Y 361.429,Z 284.311,A -85,B 0,C 180,E1 -13573.588,E2 -13573.588} C_VEL
LIN {X 0,Y 362.718,Z 209.129,A -85,B 0,C 180,E1 -13575.161,E2 -13575.161} C_VEL
LIN {X 0,Y 357.738,Z 181.962,A -85,B 0,C 180,E1 -13576.076,E2 -13576.076} C_VEL
LIN {X 0,Y 357.069,Z 176.594,A -85,B 0,C 180,E1 -13577.497,E2 -13577.497} C_VEL
LIN {X 0,Y 355.033,Z 165.901,A -85,B 0,C 180,E1 -13580.602,E2 -13580.602} C_VEL
LIN {X 0,Y 355.124,Z 165.746,A -85,B 0,C 180,E1 -13583.182,E2 -13583.182} C_VEL
LIN {X 0,Y 355.241,Z 165.737,A -85,B 0,C 180,E1 -13587.734,E2 -13587.734} C_VEL
LIN {X 0,Y 355.393,Z 165.716,A -85,B 0,C 180,E1 -13590.001,E2 -13590.001} C_VEL
LIN {X 0,Y 355.241,Z 165.732,A -85,B 0,C 180,E1 -13592.269,E2 -13592.269} C_VEL
LIN {X 0,Y 355.11,Z 165.748,A -85,B 0,C 180,E1 -13596.821,E2 -13596.821} C_VEL
LIN {X 0,Y 354.955,Z 165.767,A -85,B 0,C 180,E1 -13600.266,E2 -13600.266} C_VEL
LIN {X 0,Y 354.932,Z 165.771,A -85,B 0,C 180,E1 -13603.502,E2 -13603.502} C_VEL
LIN {X 0,Y 354.319,Z 165.852,A -85,B 0,C 180,E1 -13604.449,E2 -13604.449} C_VEL
LIN {X 0,Y 351.498,Z 166.202,A -85,B 0,C 180,E1 -13605.988,E2 -13605.988} C_VEL
LIN {X 0,Y 349.056,Z 166.506,A -85,B 0,C 180,E1 -13607.234,E2 -13607.234} C_VEL
LIN {X 0,Y 347.973,Z 166.637,A -85,B 0,C 180,E1 -13608.198,E2 -13608.198} C_VEL
LIN {X 0,Y 347.869,Z 166.65,A -85,B 0,C 180,E1 -13608.525,E2 -13608.525} C_VEL
LIN {X 0,Y 347.788,Z 166.662,A -85,B 0,C 180,E1 -13611.636,E2 -13611.636} C_VEL
LIN {X 0,Y 347.812,Z 166.662,A -85,B 0,C 180,E1 -13615.109,E2 -13615.109} C_VEL
LIN {X 0,Y 347.808,Z 166.658,A -85,B 0,C 180,E1 -13617.695,E2 -13617.695} C_VEL
LIN {X 0,Y 347.749,Z 166.665,A -85,B 0,C 180,E1 -13620.349,E2 -13620.349} C_VEL
LIN {X 0,Y 347.748,Z 166.665,A -85,B 0,C 180,E1 -13624.045,E2 -13624.045} C_VEL
LIN {X 0,Y 347.761,Z 166.665,A -85,B 0,C 180,E1 -13627.322,E2 -13627.322} C_VEL
LIN {X 0,Y 347.732,Z 166.668,A -85,B 0,C 180,E1 -13630.298,E2 -13630.298} C_VEL
LIN {X 0,Y 347.727,Z 166.668,A -85,B 0,C 180,E1 -13633.408,E2 -13633.408} C_VEL
LIN {X 0,Y 347.725,Z 166.673,A -85,B 0,C 180,E1 -13636.687,E2 -13636.687} C_VEL
LIN {X 0,Y 347.727,Z 166.669,A -85,B 0,C 180,E1 -13640.178,E2 -13640.178} C_VEL
LIN {X 0,Y 347.757,Z 166.669,A -85,B 0,C 180,E1 -13642.679,E2 -13642.679} C_VEL
LIN {X 0,Y 347.749,Z 166.666,A -85,B 0,C 180,E1 -13645.957,E2 -13645.957} C_VEL
LIN {X 0,Y 347.739,Z 166.666,A -85,B 0,C 180,E1 -13649.652,E2 -13649.652} C_VEL
LIN {X 0,Y 347.755,Z 166.664,A -85,B 0,C 180,E1 -13653.602,E2 -13653.602} C_VEL
LIN {X 0,Y 347.776,Z 166.666,A -85,B 0,C 180,E1 -13656.162,E2 -13656.162} C_VEL
LIN {X 0,Y 347.808,Z 166.66,A -85,B 0,C 180,E1 -13659.91,E2 -13659.91} C_VEL
LIN {X 0,Y 347.867,Z 166.654,A -85,B 0,C 180,E1 -13662.36,E2 -13662.36} C_VEL
LIN {X 0,Y 347.899,Z 166.651,A -85,B 0,C 180,E1 -13665.971,E2 -13665.971} C_VEL
LIN {X 0,Y 347.896,Z 166.648,A -85,B 0,C 180,E1 -13669.525,E2 -13669.525} C_VEL
LIN {X 0,Y 348.055,Z 166.626,A -85,B 0,C 180,E1 -13673.042,E2 -13673.042} C_VEL
LIN {X 0,Y 348.189,Z 166.614,A -85,B 0,C 180,E1 -13677.687,E2 -13677.687} C_VEL
LIN {X 0,Y 348.118,Z 166.62,A -85,B 0,C 180,E1 -13681.157,E2 -13681.157} C_VEL
LIN {X 0,Y 348.194,Z 166.61,A -85,B 0,C 180,E1 -13682.314,E2 -13682.314} C_VEL
LIN {X 0,Y 348.052,Z 166.627,A -85,B 0,C 180,E1 -13686.959,E2 -13686.959} C_VEL
LIN {X 0,Y 347.895,Z 166.646,A -85,B 0,C 180,E1 -13690.476,E2 -13690.476} C_VEL
LIN {X 0,Y 347.902,Z 166.646,A -85,B 0,C 180,E1 -13694.15,E2 -13694.15} C_VEL
LIN {X 0,Y 347.833,Z 166.658,A -85,B 0,C 180,E1 -13697.643,E2 -13697.643} C_VEL
LIN {X 0,Y 347.766,Z 166.665,A -85,B 0,C 180,E1 -13701.624,E2 -13701.624} C_VEL
LIN {X 0,Y 347.739,Z 166.671,A -85,B 0,C 180,E1 -13705.115,E2 -13705.115} C_VEL
LIN {X 0,Y 347.727,Z 166.669,A -85,B 0,C 180,E1 -13707.702,E2 -13707.702} C_VEL
LIN {X 0,Y 347.732,Z 166.667,A -85,B 0,C 180,E1 -13710.35,E2 -13710.35} C_VEL
LIN {X 0,Y 347.752,Z 166.664,A -85,B 0,C 180,E1 -13714.044,E2 -13714.044} C_VEL
LIN {X 0,Y 347.757,Z 166.666,A -85,B 0,C 180,E1 -13717.322,E2 -13717.322} C_VEL
LIN {X 0,Y 347.699,Z 166.672,A -85,B 0,C 180,E1 -13720.302,E2 -13720.302} C_VEL
LIN {X 0,Y 347.724,Z 166.669,A -85,B 0,C 180,E1 -13723.409,E2 -13723.409} C_VEL
LIN {X 0,Y 347.726,Z 166.673,A -85,B 0,C 180,E1 -13726.687,E2 -13726.687} C_VEL
LIN {X 0,Y 347.704,Z 166.672,A -85,B 0,C 180,E1 -13730.182,E2 -13730.182} C_VEL
LIN {X 0,Y 347.755,Z 166.67,A -85,B 0,C 180,E1 -13732.677,E2 -13732.677} C_VEL
LIN {X 0,Y 347.751,Z 166.665,A -85,B 0,C 180,E1 -13735.956,E2 -13735.956} C_VEL
LIN {X 0,Y 347.733,Z 166.672,A -85,B 0,C 180,E1 -13739.65,E2 -13739.65} C_VEL
LIN {X 0,Y 347.82,Z 166.884,A -85,B 0,C 180,E1 -13740.769,E2 -13740.769} C_VEL
LIN {X 0,Y 350.489,Z 180.068,A -85,B 0,C 180,E1 -13744.468,E2 -13744.468} C_VEL
LIN {X 0,Y 351.317,Z 186.209,A -85,B 0,C 180,E1 -13746.102,E2 -13746.102} C_VEL
LIN {X 0,Y 350.683,Z 192.306,A -85,B 0,C 180,E1 -13747.555,E2 -13747.555} C_VEL
LIN {X 0,Y 355.933,Z 224.985,A -85,B 0,C 180,E1 -13748.624,E2 -13748.624} C_VEL
LIN {X 0,Y 354.42,Z 300.637,A -85,B 0,C 180,E1 -13750.261,E2 -13750.261} C_VEL
LIN {X 0,Y 353.755,Z 314.244,A -85,B 0,C 180,E1 -13750.788,E2 -13750.788} C_VEL
LIN {X 0,Y 352.895,Z 326.601,A -85,B 0,C 180,E1 -13751.493,E2 -13751.493} C_VEL
LIN {X 0,Y 351.875,Z 338.487,A -85,B 0,C 180,E1 -13752.416,E2 -13752.416} C_VEL
LIN {X 0,Y 350.786,Z 349.939,A -85,B 0,C 180,E1 -13753.56,E2 -13753.56} C_VEL
LIN {X 0,Y 349.867,Z 360.282,A -85,B 0,C 180,E1 -13754.861,E2 -13754.861} C_VEL
LIN {X 0,Y 348.888,Z 369.552,A -85,B 0,C 180,E1 -13756.308,E2 -13756.308} C_VEL
LIN {X 0,Y 347.841,Z 378.564,A -85,B 0,C 180,E1 -13758.047,E2 -13758.047} C_VEL
LIN {X 0,Y 347.153,Z 385.807,A -85,B 0,C 180,E1 -13759.796,E2 -13759.796} C_VEL
LIN {X 0,Y 346.722,Z 390.687,A -85,B 0,C 180,E1 -13761.255,E2 -13761.255} C_VEL
LIN {X 0,Y 346.346,Z 395.411,A -85,B 0,C 180,E1 -13763.006,E2 -13763.006} C_VEL
LIN {X 0,Y 346.183,Z 398.564,A -85,B 0,C 180,E1 -13764.521,E2 -13764.521} C_VEL
LIN {X 0,Y 346.124,Z 401.559,A -85,B 0,C 180,E1 -13766.507,E2 -13766.507} C_VEL
LIN {X 0,Y 346.05,Z 402.747,A -85,B 0,C 180,E1 -13767.671,E2 -13767.671} C_VEL
LIN {X 0,Y 346.053,Z 403.485,A -85,B 0,C 180,E1 -13768.835,E2 -13768.835} C_VEL
LIN {X 0,Y 346.093,Z 403.827,A -85,B 0,C 180,E1 -13769.999,E2 -13769.999} C_VEL
LIN {X 0,Y 346.052,Z 403.776,A -85,B 0,C 180,E1 -13771.162,E2 -13771.162} C_VEL
LIN {X 0,Y 346.049,Z 403.328,A -85,B 0,C 180,E1 -13772.327,E2 -13772.327} C_VEL
LIN {X 0,Y 346.13,Z 402.439,A -85,B 0,C 180,E1 -13773.491,E2 -13773.491} C_VEL
LIN {X 0,Y 346.211,Z 401.149,A -85,B 0,C 180,E1 -13774.656,E2 -13774.656} C_VEL
LIN {X 0,Y 346.28,Z 399.145,A -85,B 0,C 180,E1 -13776.014,E2 -13776.014} C_VEL
LIN {X 0,Y 346.658,Z 394.667,A -85,B 0,C 180,E1 -13778.157,E2 -13778.157} C_VEL
LIN {X 0,Y 347.159,Z 389.793,A -85,B 0,C 180,E1 -13779.907,E2 -13779.907} C_VEL
LIN {X 0,Y 347.884,Z 383.653,A -85,B 0,C 180,E1 -13781.654,E2 -13781.654} C_VEL
LIN {X 0,Y 348.999,Z 376.028,A -85,B 0,C 180,E1 -13783.389,E2 -13783.389} C_VEL
LIN {X 0,Y 350.073,Z 368.243,A -85,B 0,C 180,E1 -13784.829,E2 -13784.829} C_VEL
LIN {X 0,Y 351.159,Z 358.765,A -85,B 0,C 180,E1 -13786.27,E2 -13786.27} C_VEL
LIN {X 0,Y 352.442,Z 348.289,A -85,B 0,C 180,E1 -13787.553,E2 -13787.553} C_VEL
LIN {X 0,Y 353.563,Z 338.25,A -85,B 0,C 180,E1 -13788.543,E2 -13788.543} C_VEL
LIN {X 0,Y 354.737,Z 326.529,A -85,B 0,C 180,E1 -13789.455,E2 -13789.455} C_VEL
LIN {X 0,Y 355.787,Z 313.723,A -85,B 0,C 180,E1 -13790.184,E2 -13790.184} C_VEL
LIN {X 0,Y 356.577,Z 300.28,A -85,B 0,C 180,E1 -13790.702,E2 -13790.702} C_VEL
LIN {X 0,Y 358.282,Z 225.333,A -85,B 0,C 180,E1 -13792.355,E2 -13792.355} C_VEL
LIN {X 0,Y 354.495,Z 203.763,A -85,B 0,C 180,E1 -13793.162,E2 -13793.162} C_VEL
LIN {X 0,Y 351.882,Z 191.514,A -85,B 0,C 180,E1 -13793.707,E2 -13793.707} C_VEL
LIN {X 0,Y 352.191,Z 188.436,A -85,B 0,C 180,E1 -13794.428,E2 -13794.428} C_VEL
LIN {X 0,Y 350.762,Z 179.899,A -85,B 0,C 180,E1 -13796.794,E2 -13796.794} C_VEL
LIN {X 0,Y 348.065,Z 168.006,A -85,B 0,C 180,E1 -13800.316,E2 -13800.316} C_VEL
LIN {X 0,Y 347.741,Z 166.699,A -85,B 0,C 180,E1 -13800.809,E2 -13800.809} C_VEL
LIN {X 0,Y 347.738,Z 166.671,A -85,B 0,C 180,E1 -13804.462,E2 -13804.462} C_VEL
LIN {X 0,Y 347.756,Z 166.666,A -85,B 0,C 180,E1 -13807.984,E2 -13807.984} C_VEL
LIN {X 0,Y 347.734,Z 166.669,A -85,B 0,C 180,E1 -13811.83,E2 -13811.83} C_VEL
LIN {X 0,Y 347.693,Z 166.675,A -85,B 0,C 180,E1 -13815.026,E2 -13815.026} C_VEL
LIN {X 0,Y 347.73,Z 166.67,A -85,B 0,C 180,E1 -13818.398,E2 -13818.398} C_VEL
LIN {X 0,Y 347.753,Z 166.662,A -85,B 0,C 180,E1 -13822.013,E2 -13822.013} C_VEL
LIN {X 0,Y 347.734,Z 166.664,A -85,B 0,C 180,E1 -13825.534,E2 -13825.534} C_VEL
LIN {X 0,Y 347.735,Z 166.667,A -85,B 0,C 180,E1 -13828.299,E2 -13828.299} C_VEL
LIN {X 0,Y 347.734,Z 166.672,A -85,B 0,C 180,E1 -13830.983,E2 -13830.983} C_VEL
LIN {X 0,Y 347.756,Z 166.67,A -85,B 0,C 180,E1 -13834.887,E2 -13834.887} C_VEL
LIN {X 0,Y 347.769,Z 166.665,A -85,B 0,C 180,E1 -13838.668,E2 -13838.668} C_VEL
LIN {X 0,Y 347.832,Z 166.654,A -85,B 0,C 180,E1 -13842.357,E2 -13842.357} C_VEL
LIN {X 0,Y 347.887,Z 166.647,A -85,B 0,C 180,E1 -13845.97,E2 -13845.97} C_VEL
LIN {X 0,Y 347.883,Z 166.647,A -85,B 0,C 180,E1 -13849.524,E2 -13849.524} C_VEL
LIN {X 0,Y 348.06,Z 166.623,A -85,B 0,C 180,E1 -13853.041,E2 -13853.041} C_VEL
LIN {X 0,Y 348.18,Z 166.611,A -85,B 0,C 180,E1 -13857.686,E2 -13857.686} C_VEL
LIN {X 0,Y 348.13,Z 166.62,A -85,B 0,C 180,E1 -13861.156,E2 -13861.156} C_VEL
LIN {X 0,Y 348.176,Z 166.615,A -85,B 0,C 180,E1 -13862.313,E2 -13862.313} C_VEL
LIN {X 0,Y 348.059,Z 166.628,A -85,B 0,C 180,E1 -13866.958,E2 -13866.958} C_VEL
LIN {X 0,Y 347.878,Z 166.655,A -85,B 0,C 180,E1 -13870.475,E2 -13870.475} C_VEL
LIN {X 0,Y 347.886,Z 166.65,A -85,B 0,C 180,E1 -13874.15,E2 -13874.15} C_VEL
LIN {X 0,Y 347.816,Z 166.661,A -85,B 0,C 180,E1 -13878.259,E2 -13878.259} C_VEL
LIN {X 0,Y 347.754,Z 166.669,A -85,B 0,C 180,E1 -13881.626,E2 -13881.626} C_VEL
LIN {X 0,Y 347.773,Z 166.776,A -85,B 0,C 180,E1 -13885.672,E2 -13885.672} C_VEL
LIN {X 0,Y 350.349,Z 177.968,A -85,B 0,C 180,E1 -13889.107,E2 -13889.107} C_VEL
LIN {X 0,Y 351.233,Z 182.236,A -85,B 0,C 180,E1 -13890.278,E2 -13890.278} C_VEL
LIN {X 0,Y 354.143,Z 190.06,A -85,B 0,C 180,E1 -13890.751,E2 -13890.751} C_VEL
LIN {X 0,Y 357.778,Z 207.123,A -85,B 0,C 180,E1 -13891.451,E2 -13891.451} C_VEL
LIN {X 0,Y 358.639,Z 212.138,A -85,B 0,C 180,E1 -13891.634,E2 -13891.634} C_VEL
LIN {X 0,Y 356.652,Z 290.376,A -85,B 0,C 180,E1 -13893.348,E2 -13893.348} C_VEL
LIN {X 0,Y 355.983,Z 303.608,A -85,B 0,C 180,E1 -13893.865,E2 -13893.865} C_VEL
LIN {X 0,Y 355.09,Z 316.205,A -85,B 0,C 180,E1 -13894.589,E2 -13894.589} C_VEL
LIN {X 0,Y 353.992,Z 328.068,A -85,B 0,C 180,E1 -13895.515,E2 -13895.515} C_VEL
LIN {X 0,Y 352.69,Z 339.937,A -85,B 0,C 180,E1 -13896.712,E2 -13896.712} C_VEL
LIN {X 0,Y 351.443,Z 349.622,A -85,B 0,C 180,E1 -13897.934,E2 -13897.934} C_VEL
LIN {X 0,Y 350.259,Z 358.794,A -85,B 0,C 180,E1 -13899.369,E2 -13899.369} C_VEL
LIN {X 0,Y 349.123,Z 367.211,A -85,B 0,C 180,E1 -13900.988,E2 -13900.988} C_VEL
LIN {X 0,Y 348.205,Z 373.839,A -85,B 0,C 180,E1 -13902.552,E2 -13902.552} C_VEL
LIN {X 0,Y 347.343,Z 380.509,A -85,B 0,C 180,E1 -13904.523,E2 -13904.523} C_VEL
LIN {X 0,Y 346.757,Z 385.446,A -85,B 0,C 180,E1 -13906.443,E2 -13906.443} C_VEL
LIN {X 0,Y 346.335,Z 389.533,A -85,B 0,C 180,E1 -13908.661,E2 -13908.661} C_VEL
LIN {X 0,Y 345.966,Z 392.141,A -85,B 0,C 180,E1 -13910.972,E2 -13910.972} C_VEL
LIN {X 0,Y 345.864,Z 392.947,A -85,B 0,C 180,E1 -13912.441,E2 -13912.441} C_VEL
LIN {X 0,Y 345.831,Z 393.043,A -85,B 0,C 180,E1 -13914.378,E2 -13914.378} C_VEL
LIN {X 0,Y 345.889,Z 391.946,A -85,B 0,C 180,E1 -13916.414,E2 -13916.414} C_VEL
LIN {X 0,Y 346.137,Z 389.461,A -85,B 0,C 180,E1 -13918.513,E2 -13918.513} C_VEL
LIN {X 0,Y 346.459,Z 385.341,A -85,B 0,C 180,E1 -13920.722,E2 -13920.722} C_VEL
LIN {X 0,Y 346.934,Z 380.282,A -85,B 0,C 180,E1 -13922.662,E2 -13922.662} C_VEL
LIN {X 0,Y 347.523,Z 373.838,A -85,B 0,C 180,E1 -13924.551,E2 -13924.551} C_VEL
LIN {X 0,Y 348.215,Z 366.826,A -85,B 0,C 180,E1 -13926.195,E2 -13926.195} C_VEL
LIN {X 0,Y 349.212,Z 357.776,A -85,B 0,C 180,E1 -13927.906,E2 -13927.906} C_VEL
LIN {X 0,Y 350.299,Z 347.498,A -85,B 0,C 180,E1 -13929.447,E2 -13929.447} C_VEL
LIN {X 0,Y 351.426,Z 336.772,A -85,B 0,C 180,E1 -13930.734,E2 -13930.734} C_VEL
LIN {X 0,Y 352.45,Z 325.017,A -85,B 0,C 180,E1 -13931.848,E2 -13931.848} C_VEL
LIN {X 0,Y 353.297,Z 313.113,A -85,B 0,C 180,E1 -13932.714,E2 -13932.714} C_VEL
LIN {X 0,Y 354.049,Z 300.575,A -85,B 0,C 180,E1 -13933.385,E2 -13933.385} C_VEL
LIN {X 0,Y 354.554,Z 288.604,A -85,B 0,C 180,E1 -13933.816,E2 -13933.816} C_VEL
LIN {X 0,Y 356.017,Z 210.074,A -85,B 0,C 180,E1 -13935.506,E2 -13935.506} C_VEL
LIN {X 0,Y 351.075,Z 183.467,A -85,B 0,C 180,E1 -13936.397,E2 -13936.397} C_VEL
LIN {X 0,Y 350.736,Z 181.804,A -85,B 0,C 180,E1 -13936.531,E2 -13936.531} C_VEL
LIN {X 0,Y 349.175,Z 173.13,A -85,B 0,C 180,E1 -13938.978,E2 -13938.978} C_VEL
LIN {X 0,Y 347.998,Z 166.73,A -85,B 0,C 180,E1 -13940.924,E2 -13940.924} C_VEL
LIN {X 0,Y 348.061,Z 166.628,A -85,B 0,C 180,E1 -13944.207,E2 -13944.207} C_VEL
LIN {X 0,Y 348.203,Z 166.613,A -85,B 0,C 180,E1 -13947.688,E2 -13947.688} C_VEL
LIN {X 0,Y 348.342,Z 166.594,A -85,B 0,C 180,E1 -13950.001,E2 -13950.001} C_VEL
LIN {X 0,Y 348.204,Z 166.609,A -85,B 0,C 180,E1 -13952.315,E2 -13952.315} C_VEL
LIN {X 0,Y 348.076,Z 166.625,A -85,B 0,C 180,E1 -13956.959,E2 -13956.959} C_VEL
LIN {X 0,Y 347.895,Z 166.646,A -85,B 0,C 180,E1 -13960.476,E2 -13960.476} C_VEL
LIN {X 0,Y 347.897,Z 166.647,A -85,B 0,C 180,E1 -13964.151,E2 -13964.151} C_VEL
LIN {X 0,Y 347.89,Z 166.647,A -85,B 0,C 180,E1 -13968.291,E2 -13968.291} C_VEL
LIN {X 0,Y 347.869,Z 166.65,A -85,B 0,C 180,E1 -13968.525,E2 -13968.525} C_VEL
LIN {X 0,Y 347.148,Z 166.744,A -85,B 0,C 180,E1 -13969.491,E2 -13969.491} C_VEL
LIN {X 0,Y 344.244,Z 167.107,A -85,B 0,C 180,E1 -13971.063,E2 -13971.063} C_VEL
LIN {X 0,Y 341.821,Z 167.407,A -85,B 0,C 180,E1 -13972.335,E2 -13972.335} C_VEL
LIN {X 0,Y 340.796,Z 167.536,A -85,B 0,C 180,E1 -13973.32,E2 -13973.32} C_VEL
LIN {X 0,Y 340.719,Z 167.54,A -85,B 0,C 180,E1 -13973.654,E2 -13973.654} C_VEL
LIN {X 0,Y 340.803,Z 167.533,A -85,B 0,C 180,E1 -13976.981,E2 -13976.981} C_VEL
LIN {X 0,Y 340.697,Z 167.549,A -85,B 0,C 180,E1 -13981.046,E2 -13981.046} C_VEL
LIN {X 0,Y 340.718,Z 167.542,A -85,B 0,C 180,E1 -13985.28,E2 -13985.28} C_VEL
LIN {X 0,Y 340.709,Z 167.542,A -85,B 0,C 180,E1 -13988.387,E2 -13988.387} C_VEL
LIN {X 0,Y 340.699,Z 167.543,A -85,B 0,C 180,E1 -13992.046,E2 -13992.046} C_VEL
LIN {X 0,Y 340.682,Z 167.545,A -85,B 0,C 180,E1 -13995.462,E2 -13995.462} C_VEL
LIN {X 0,Y 340.68,Z 167.549,A -85,B 0,C 180,E1 -13998.69,E2 -13998.69} C_VEL
LIN {X 0,Y 340.719,Z 167.54,A -85,B 0,C 180,E1 -14001.772,E2 -14001.772} C_VEL
LIN {X 0,Y 340.723,Z 167.54,A -85,B 0,C 180,E1 -14005.596,E2 -14005.596} C_VEL
LIN {X 0,Y 340.694,Z 167.545,A -85,B 0,C 180,E1 -14008.956,E2 -14008.956} C_VEL
LIN {X 0,Y 340.724,Z 167.541,A -85,B 0,C 180,E1 -14013.014,E2 -14013.014} C_VEL
LIN {X 0,Y 340.745,Z 167.538,A -85,B 0,C 180,E1 -14015.638,E2 -14015.638} C_VEL
LIN {X 0,Y 340.737,Z 167.538,A -85,B 0,C 180,E1 -14019.474,E2 -14019.474} C_VEL
LIN {X 0,Y 340.859,Z 167.527,A -85,B 0,C 180,E1 -14021.985,E2 -14021.985} C_VEL
LIN {X 0,Y 340.871,Z 167.523,A -85,B 0,C 180,E1 -14025.706,E2 -14025.706} C_VEL
LIN {X 0,Y 340.848,Z 167.525,A -85,B 0,C 180,E1 -14029.306,E2 -14029.306} C_VEL
LIN {X 0,Y 341.002,Z 167.505,A -85,B 0,C 180,E1 -14032.897,E2 -14032.897} C_VEL
LIN {X 0,Y 340.813,Z 167.529,A -85,B 0,C 180,E1 -14035.269,E2 -14035.269} C_VEL
LIN {X 0,Y 341.126,Z 167.494,A -85,B 0,C 180,E1 -14037.639,E2 -14037.639} C_VEL
LIN {X 0,Y 341.089,Z 167.494,A -85,B 0,C 180,E1 -14041.181,E2 -14041.181} C_VEL
LIN {X 0,Y 341.131,Z 167.488,A -85,B 0,C 180,E1 -14042.362,E2 -14042.362} C_VEL
LIN {X 0,Y 341,Z 167.506,A -85,B 0,C 180,E1 -14047.104,E2 -14047.104} C_VEL
LIN {X 0,Y 340.848,Z 167.524,A -85,B 0,C 180,E1 -14050.695,E2 -14050.695} C_VEL
LIN {X 0,Y 340.867,Z 167.521,A -85,B 0,C 180,E1 -14054.325,E2 -14054.325} C_VEL
LIN {X 0,Y 340.773,Z 167.533,A -85,B 0,C 180,E1 -14058.432,E2 -14058.432} C_VEL
LIN {X 0,Y 340.721,Z 167.541,A -85,B 0,C 180,E1 -14061.842,E2 -14061.842} C_VEL
LIN {X 0,Y 340.672,Z 167.547,A -85,B 0,C 180,E1 -14065.673,E2 -14065.673} C_VEL
LIN {X 0,Y 340.678,Z 167.545,A -85,B 0,C 180,E1 -14068.326,E2 -14068.326} C_VEL
LIN {X 0,Y 340.685,Z 167.55,A -85,B 0,C 180,E1 -14071.047,E2 -14071.047} C_VEL
LIN {X 0,Y 340.718,Z 167.544,A -85,B 0,C 180,E1 -14075.279,E2 -14075.279} C_VEL
LIN {X 0,Y 340.696,Z 167.544,A -85,B 0,C 180,E1 -14078.382,E2 -14078.382} C_VEL
LIN {X 0,Y 340.694,Z 167.544,A -85,B 0,C 180,E1 -14082.044,E2 -14082.044} C_VEL
LIN {X 0,Y 340.653,Z 167.55,A -85,B 0,C 180,E1 -14086.227,E2 -14086.227} C_VEL
LIN {X 0,Y 340.672,Z 167.552,A -85,B 0,C 180,E1 -14088.688,E2 -14088.688} C_VEL
LIN {X 0,Y 340.72,Z 167.54,A -85,B 0,C 180,E1 -14091.77,E2 -14091.77} C_VEL
LIN {X 0,Y 340.723,Z 167.54,A -85,B 0,C 180,E1 -14095.596,E2 -14095.596} C_VEL
LIN {X 0,Y 340.685,Z 167.549,A -85,B 0,C 180,E1 -14098.953,E2 -14098.953} C_VEL
LIN {X 0,Y 340.728,Z 167.684,A -85,B 0,C 180,E1 -14100.412,E2 -14100.412} C_VEL
LIN {X 0,Y 343.146,Z 179.357,A -85,B 0,C 180,E1 -14103.791,E2 -14103.791} C_VEL
LIN {X 0,Y 344.359,Z 187.094,A -85,B 0,C 180,E1 -14105.909,E2 -14105.909} C_VEL
LIN {X 0,Y 343.802,Z 192.054,A -85,B 0,C 180,E1 -14107.12,E2 -14107.12} C_VEL
LIN {X 0,Y 344.874,Z 198.697,A -85,B 0,C 180,E1 -14107.39,E2 -14107.39} C_VEL
LIN {X 0,Y 349.244,Z 226.246,A -85,B 0,C 180,E1 -14108.283,E2 -14108.283} C_VEL
LIN {X 0,Y 347.686,Z 299.925,A -85,B 0,C 180,E1 -14109.901,E2 -14109.901} C_VEL
LIN {X 0,Y 346.987,Z 313.716,A -85,B 0,C 180,E1 -14110.437,E2 -14110.437} C_VEL
LIN {X 0,Y 346.04,Z 326.718,A -85,B 0,C 180,E1 -14111.19,E2 -14111.19} C_VEL
LIN {X 0,Y 344.936,Z 339.347,A -85,B 0,C 180,E1 -14112.203,E2 -14112.203} C_VEL
LIN {X 0,Y 343.822,Z 350.625,A -85,B 0,C 180,E1 -14113.37,E2 -14113.37} C_VEL
LIN {X 0,Y 342.868,Z 360.782,A -85,B 0,C 180,E1 -14114.697,E2 -14114.697} C_VEL
LIN {X 0,Y 341.788,Z 370.772,A -85,B 0,C 180,E1 -14116.321,E2 -14116.321} C_VEL
LIN {X 0,Y 340.699,Z 379.544,A -85,B 0,C 180,E1 -14118.094,E2 -14118.094} C_VEL
LIN {X 0,Y 340.019,Z 386.532,A -85,B 0,C 180,E1 -14119.88,E2 -14119.88} C_VEL
LIN {X 0,Y 339.533,Z 392.119,A -85,B 0,C 180,E1 -14121.668,E2 -14121.668} C_VEL
LIN {X 0,Y 339.23,Z 396.486,A -85,B 0,C 180,E1 -14123.456,E2 -14123.456} C_VEL
LIN {X 0,Y 339.062,Z 399.759,A -85,B 0,C 180,E1 -14125.243,E2 -14125.243} C_VEL
LIN {X 0,Y 339.05,Z 401.383,A -85,B 0,C 180,E1 -14126.434,E2 -14126.434} C_VEL
LIN {X 0,Y 338.967,Z 402.593,A -85,B 0,C 180,E1 -14127.622,E2 -14127.622} C_VEL
LIN {X 0,Y 338.959,Z 403.353,A -85,B 0,C 180,E1 -14128.811,E2 -14128.811} C_VEL
LIN {X 0,Y 338.995,Z 403.709,A -85,B 0,C 180,E1 -14129.999,E2 -14129.999} C_VEL
LIN {X 0,Y 338.958,Z 403.672,A -85,B 0,C 180,E1 -14131.187,E2 -14131.187} C_VEL
LIN {X 0,Y 338.966,Z 403.243,A -85,B 0,C 180,E1 -14132.375,E2 -14132.375} C_VEL
LIN {X 0,Y 339.059,Z 402.375,A -85,B 0,C 180,E1 -14133.564,E2 -14133.564} C_VEL
LIN {X 0,Y 339.114,Z 401.098,A -85,B 0,C 180,E1 -14134.754,E2 -14134.754} C_VEL
LIN {X 0,Y 339.253,Z 398.396,A -85,B 0,C 180,E1 -14136.54,E2 -14136.54} C_VEL
LIN {X 0,Y 339.606,Z 394.67,A -85,B 0,C 180,E1 -14138.328,E2 -14138.328} C_VEL
LIN {X 0,Y 340.144,Z 389.824,A -85,B 0,C 180,E1 -14140.114,E2 -14140.114} C_VEL
LIN {X 0,Y 340.902,Z 383.724,A -85,B 0,C 180,E1 -14141.896,E2 -14141.896} C_VEL
LIN {X 0,Y 342.094,Z 376.152,A -85,B 0,C 180,E1 -14143.664,E2 -14143.664} C_VEL
LIN {X 0,Y 343.208,Z 368.434,A -85,B 0,C 180,E1 -14145.133,E2 -14145.133} C_VEL
LIN {X 0,Y 344.176,Z 360.484,A -85,B 0,C 180,E1 -14146.397,E2 -14146.397} C_VEL
LIN {X 0,Y 345.572,Z 349.944,A -85,B 0,C 180,E1 -14147.76,E2 -14147.76} C_VEL
LIN {X 0,Y 346.861,Z 338.725,A -85,B 0,C 180,E1 -14148.915,E2 -14148.915} C_VEL
LIN {X 0,Y 348.212,Z 326.155,A -85,B 0,C 180,E1 -14149.911,E2 -14149.911} C_VEL
LIN {X 0,Y 349.257,Z 313.242,A -85,B 0,C 180,E1 -14150.656,E2 -14150.656} C_VEL
LIN {X 0,Y 350.098,Z 299.639,A -85,B 0,C 180,E1 -14151.181,E2 -14151.181} C_VEL
LIN {X 0,Y 351.853,Z 226.168,A -85,B 0,C 180,E1 -14152.828,E2 -14152.828} C_VEL
LIN {X 0,Y 348.14,Z 205.001,A -85,B 0,C 180,E1 -14153.652,E2 -14153.652} C_VEL
LIN {X 0,Y 345.243,Z 191.416,A -85,B 0,C 180,E1 -14154.275,E2 -14154.275} C_VEL
LIN {X 0,Y 345.185,Z 188.509,A -85,B 0,C 180,E1 -14154.989,E2 -14154.989} C_VEL
LIN {X 0,Y 343.574,Z 180.12,A -85,B 0,C 180,E1 -14157.401,E2 -14157.401} C_VEL
LIN {X 0,Y 341.293,Z 170.027,A -85,B 0,C 180,E1 -14160.48,E2 -14160.48} C_VEL
LIN {X 0,Y 340.698,Z 167.575,A -85,B 0,C 180,E1 -14161.345,E2 -14161.345} C_VEL
LIN {X 0,Y 340.711,Z 167.546,A -85,B 0,C 180,E1 -14165.278,E2 -14165.278} C_VEL
LIN {X 0,Y 340.688,Z 167.546,A -85,B 0,C 180,E1 -14168.38,E2 -14168.38} C_VEL
LIN {X 0,Y 340.684,Z 167.547,A -85,B 0,C 180,E1 -14172.042,E2 -14172.042} C_VEL
LIN {X 0,Y 340.642,Z 167.552,A -85,B 0,C 180,E1 -14176.226,E2 -14176.226} C_VEL
LIN {X 0,Y 340.661,Z 167.552,A -85,B 0,C 180,E1 -14178.686,E2 -14178.686} C_VEL
LIN {X 0,Y 340.71,Z 167.54,A -85,B 0,C 180,E1 -14181.769,E2 -14181.769} C_VEL
LIN {X 0,Y 340.713,Z 167.538,A -85,B 0,C 180,E1 -14185.594,E2 -14185.594} C_VEL
LIN {X 0,Y 340.682,Z 167.542,A -85,B 0,C 180,E1 -14188.953,E2 -14188.953} C_VEL
LIN {X 0,Y 340.701,Z 167.539,A -85,B 0,C 180,E1 -14193.011,E2 -14193.011} C_VEL
LIN {X 0,Y 340.729,Z 167.539,A -85,B 0,C 180,E1 -14195.636,E2 -14195.636} C_VEL
LIN {X 0,Y 340.717,Z 167.54,A -85,B 0,C 180,E1 -14199.472,E2 -14199.472} C_VEL
LIN {X 0,Y 340.781,Z 167.531,A -85,B 0,C 180,E1 -14201.98,E2 -14201.98} C_VEL
LIN {X 0,Y 340.859,Z 167.522,A -85,B 0,C 180,E1 -14205.704,E2 -14205.704} C_VEL
LIN {X 0,Y 340.835,Z 167.523,A -85,B 0,C 180,E1 -14209.305,E2 -14209.305} C_VEL
LIN {X 0,Y 341.007,Z 167.501,A -85,B 0,C 180,E1 -14212.896,E2 -14212.896} C_VEL
LIN {X 0,Y 340.813,Z 167.529,A -85,B 0,C 180,E1 -14215.268,E2 -14215.268} C_VEL
LIN {X 0,Y 341.117,Z 167.491,A -85,B 0,C 180,E1 -14217.638,E2 -14217.638} C_VEL
LIN {X 0,Y 341.098,Z 167.496,A -85,B 0,C 180,E1 -14221.18,E2 -14221.18} C_VEL
LIN {X 0,Y 341.113,Z 167.494,A -85,B 0,C 180,E1 -14222.361,E2 -14222.361} C_VEL
LIN {X 0,Y 341.028,Z 167.505,A -85,B 0,C 180,E1 -14227.102,E2 -14227.102} C_VEL
LIN {X 0,Y 340.831,Z 167.53,A -85,B 0,C 180,E1 -14230.695,E2 -14230.695} C_VEL
LIN {X 0,Y 340.851,Z 167.526,A -85,B 0,C 180,E1 -14234.325,E2 -14234.325} C_VEL
LIN {X 0,Y 340.773,Z 167.539,A -85,B 0,C 180,E1 -14238.44,E2 -14238.44} C_VEL
LIN {X 0,Y 340.705,Z 167.547,A -85,B 0,C 180,E1 -14241.842,E2 -14241.842} C_VEL
LIN {X 0,Y 340.714,Z 167.719,A -85,B 0,C 180,E1 -14245.184,E2 -14245.184} C_VEL
LIN {X 0,Y 343.381,Z 179.055,A -85,B 0,C 180,E1 -14248.748,E2 -14248.748} C_VEL
LIN {X 0,Y 344.117,Z 182.465,A -85,B 0,C 180,E1 -14249.687,E2 -14249.687} C_VEL
LIN {X 0,Y 348.107,Z 192.655,A -85,B 0,C 180,E1 -14250.313,E2 -14250.313} C_VEL
LIN {X 0,Y 351.609,Z 209.447,A -85,B 0,C 180,E1 -14251.021,E2 -14251.021} C_VEL
LIN {X 0,Y 352.2,Z 213.899,A -85,B 0,C 180,E1 -14251.178,E2 -14251.178} C_VEL
LIN {X 0,Y 350.181,Z 290.35,A -85,B 0,C 180,E1 -14252.885,E2 -14252.885} C_VEL
LIN {X 0,Y 349.473,Z 303.417,A -85,B 0,C 180,E1 -14253.399,E2 -14253.399} C_VEL
LIN {X 0,Y 348.562,Z 315.818,A -85,B 0,C 180,E1 -14254.116,E2 -14254.116} C_VEL
LIN {X 0,Y 347.493,Z 327.257,A -85,B 0,C 180,E1 -14255.008,E2 -14255.008} C_VEL
LIN {X 0,Y 346.154,Z 338.738,A -85,B 0,C 180,E1 -14256.16,E2 -14256.16} C_VEL
LIN {X 0,Y 344.883,Z 348.423,A -85,B 0,C 180,E1 -14257.373,E2 -14257.373} C_VEL
LIN {X 0,Y 343.645,Z 357.51,A -85,B 0,C 180,E1 -14258.769,E2 -14258.769} C_VEL
LIN {X 0,Y 342.293,Z 366.873,A -85,B 0,C 180,E1 -14260.566,E2 -14260.566} C_VEL
LIN {X 0,Y 341.334,Z 373.587,A -85,B 0,C 180,E1 -14262.166,E2 -14262.166} C_VEL
LIN {X 0,Y 340.375,Z 380.484,A -85,B 0,C 180,E1 -14264.23,E2 -14264.23} C_VEL
LIN {X 0,Y 339.686,Z 385.894,A -85,B 0,C 180,E1 -14266.396,E2 -14266.396} C_VEL
LIN {X 0,Y 339.278,Z 389.623,A -85,B 0,C 180,E1 -14268.484,E2 -14268.484} C_VEL
LIN {X 0,Y 338.98,Z 391.582,A -85,B 0,C 180,E1 -14270.094,E2 -14270.094} C_VEL
LIN {X 0,Y 338.762,Z 392.931,A -85,B 0,C 180,E1 -14272.031,E2 -14272.031} C_VEL
LIN {X 0,Y 338.746,Z 393.202,A -85,B 0,C 180,E1 -14274.011,E2 -14274.011} C_VEL
LIN {X 0,Y 338.765,Z 392.294,A -85,B 0,C 180,E1 -14276.081,E2 -14276.081} C_VEL
LIN {X 0,Y 339.002,Z 390.08,A -85,B 0,C 180,E1 -14278.209,E2 -14278.209} C_VEL
LIN {X 0,Y 339.334,Z 386.221,A -85,B 0,C 180,E1 -14280.442,E2 -14280.442} C_VEL
LIN {X 0,Y 339.716,Z 381.964,A -85,B 0,C 180,E1 -14282.221,E2 -14282.221} C_VEL
LIN {X 0,Y 340.319,Z 375.478,A -85,B 0,C 180,E1 -14284.301,E2 -14284.301} C_VEL
LIN {X 0,Y 341.038,Z 368.794,A -85,B 0,C 180,E1 -14285.985,E2 -14285.985} C_VEL
LIN {X 0,Y 341.931,Z 360.571,A -85,B 0,C 180,E1 -14287.655,E2 -14287.655} C_VEL
LIN {X 0,Y 343.138,Z 350.405,A -85,B 0,C 180,E1 -14289.312,E2 -14289.312} C_VEL
LIN {X 0,Y 344.211,Z 339.854,A -85,B 0,C 180,E1 -14290.686,E2 -14290.686} C_VEL
LIN {X 0,Y 345.343,Z 327.783,A -85,B 0,C 180,E1 -14291.921,E2 -14291.921} C_VEL
LIN {X 0,Y 346.316,Z 315.705,A -85,B 0,C 180,E1 -14292.876,E2 -14292.876} C_VEL
LIN {X 0,Y 347.072,Z 302.681,A -85,B 0,C 180,E1 -14293.627,E2 -14293.627} C_VEL
LIN {X 0,Y 347.767,Z 288.993,A -85,B 0,C 180,E1 -14294.151,E2 -14294.151} C_VEL
LIN {X 0,Y 349.235,Z 210.542,A -85,B 0,C 180,E1 -14295.878,E2 -14295.878} C_VEL
LIN {X 0,Y 344.232,Z 184.172,A -85,B 0,C 180,E1 -14296.779,E2 -14296.779} C_VEL
LIN {X 0,Y 343.577,Z 181.926,A -85,B 0,C 180,E1 -14296.96,E2 -14296.96} C_VEL
LIN {X 0,Y 341.689,Z 171.689,A -85,B 0,C 180,E1 -14299.933,E2 -14299.933} C_VEL
LIN {X 0,Y 340.977,Z 167.54,A -85,B 0,C 180,E1 -14301.269,E2 -14301.269} C_VEL
LIN {X 0,Y 341.037,Z 167.505,A -85,B 0,C 180,E1 -14304.087,E2 -14304.087} C_VEL
LIN {X 0,Y 341.165,Z 167.489,A -85,B 0,C 180,E1 -14307.64,E2 -14307.64} C_VEL
LIN {X 0,Y 341.292,Z 167.472,A -85,B 0,C 180,E1 -14310.001,E2 -14310.001} C_VEL
LIN {X 0,Y 341.165,Z 167.485,A -85,B 0,C 180,E1 -14312.362,E2 -14312.362} C_VEL
LIN {X 0,Y 341.043,Z 167.502,A -85,B 0,C 180,E1 -14317.104,E2 -14317.104} C_VEL
LIN {X 0,Y 340.847,Z 167.525,A -85,B 0,C 180,E1 -14320.696,E2 -14320.696} C_VEL
LIN {X 0,Y 340.862,Z 167.523,A -85,B 0,C 180,E1 -14324.326,E2 -14324.326} C_VEL
LIN {X 0,Y 340.832,Z 167.526,A -85,B 0,C 180,E1 -14328.506,E2 -14328.506} C_VEL
LIN {X 0,Y 340.753,Z 167.537,A -85,B 0,C 180,E1 -14331.858,E2 -14331.858} C_VEL
LIN {X 0,Y 340.719,Z 167.54,A -85,B 0,C 180,E1 -14333.654,E2 -14333.654} C_VEL
LIN {X 0,Y 340.064,Z 167.624,A -85,B 0,C 180,E1 -14334.64,E2 -14334.64} C_VEL
LIN {X 0,Y 337.203,Z 167.977,A -85,B 0,C 180,E1 -14336.245,E2 -14336.245} C_VEL
LIN {X 0,Y 334.782,Z 168.281,A -85,B 0,C 180,E1 -14337.544,E2 -14337.544} C_VEL
LIN {X 0,Y 333.76,Z 168.408,A -85,B 0,C 180,E1 -14338.55,E2 -14338.55} C_VEL
LIN {X 0,Y 333.687,Z 168.419,A -85,B 0,C 180,E1 -14338.891,E2 -14338.891} C_VEL
LIN {X 0,Y 333.643,Z 168.424,A -85,B 0,C 180,E1 -14342.588,E2 -14342.588} C_VEL
LIN {X 0,Y 333.676,Z 168.415,A -85,B 0,C 180,E1 -14346.14,E2 -14346.14} C_VEL
LIN {X 0,Y 333.646,Z 168.424,A -85,B 0,C 180,E1 -14349.193,E2 -14349.193} C_VEL
LIN {X 0,Y 333.633,Z 168.426,A -85,B 0,C 180,E1 -14352.501,E2 -14352.501} C_VEL
LIN {X 0,Y 333.619,Z 168.424,A -85,B 0,C 180,E1 -14355.96,E2 -14355.96} C_VEL
LIN {X 0,Y 333.642,Z 168.42,A -85,B 0,C 180,E1 -14359.317,E2 -14359.317} C_VEL
LIN {X 0,Y 333.663,Z 168.42,A -85,B 0,C 180,E1 -14363.169,E2 -14363.169} C_VEL
LIN {X 0,Y 333.674,Z 168.418,A -85,B 0,C 180,E1 -14365.342,E2 -14365.342} C_VEL
LIN {X 0,Y 333.63,Z 168.426,A -85,B 0,C 180,E1 -14368.223,E2 -14368.223} C_VEL
LIN {X 0,Y 333.654,Z 168.421,A -85,B 0,C 180,E1 -14371.023,E2 -14371.023} C_VEL
LIN {X 0,Y 333.7,Z 168.415,A -85,B 0,C 180,E1 -14375.089,E2 -14375.089} C_VEL
LIN {X 0,Y 333.675,Z 168.418,A -85,B 0,C 180,E1 -14379.019,E2 -14379.019} C_VEL
LIN {X 0,Y 333.795,Z 168.404,A -85,B 0,C 180,E1 -14381.59,E2 -14381.59} C_VEL
LIN {X 0,Y 333.81,Z 168.401,A -85,B 0,C 180,E1 -14385.577,E2 -14385.577} C_VEL
LIN {X 0,Y 333.818,Z 168.4,A -85,B 0,C 180,E1 -14389.078,E2 -14389.078} C_VEL
LIN {X 0,Y 333.958,Z 168.382,A -85,B 0,C 180,E1 -14392.747,E2 -14392.747} C_VEL
LIN {X 0,Y 333.779,Z 168.405,A -85,B 0,C 180,E1 -14395.169,E2 -14395.169} C_VEL
LIN {X 0,Y 334.066,Z 168.372,A -85,B 0,C 180,E1 -14397.589,E2 -14397.589} C_VEL
LIN {X 0,Y 334.06,Z 168.369,A -85,B 0,C 180,E1 -14401.206,E2 -14401.206} C_VEL
LIN {X 0,Y 334.071,Z 168.366,A -85,B 0,C 180,E1 -14402.412,E2 -14402.412} C_VEL
LIN {X 0,Y 333.986,Z 168.38,A -85,B 0,C 180,E1 -14406.04,E2 -14406.04} C_VEL
LIN {X 0,Y 333.916,Z 168.388,A -85,B 0,C 180,E1 -14408.473,E2 -14408.473} C_VEL
LIN {X 0,Y 333.792,Z 168.404,A -85,B 0,C 180,E1 -14412.155,E2 -14412.155} C_VEL
LIN {X 0,Y 333.811,Z 168.399,A -85,B 0,C 180,E1 -14414.635,E2 -14414.635} C_VEL
LIN {X 0,Y 333.711,Z 168.413,A -85,B 0,C 180,E1 -14418.61,E2 -14418.61} C_VEL
LIN {X 0,Y 333.652,Z 168.421,A -85,B 0,C 180,E1 -14422.282,E2 -14422.282} C_VEL
LIN {X 0,Y 333.66,Z 168.423,A -85,B 0,C 180,E1 -14425.078,E2 -14425.078} C_VEL
LIN {X 0,Y 333.651,Z 168.425,A -85,B 0,C 180,E1 -14428.978,E2 -14428.978} C_VEL
LIN {X 0,Y 333.64,Z 168.423,A -85,B 0,C 180,E1 -14432.585,E2 -14432.585} C_VEL
LIN {X 0,Y 333.676,Z 168.418,A -85,B 0,C 180,E1 -14436.14,E2 -14436.14} C_VEL
LIN {X 0,Y 333.623,Z 168.426,A -85,B 0,C 180,E1 -14439.196,E2 -14439.196} C_VEL
LIN {X 0,Y 333.63,Z 168.426,A -85,B 0,C 180,E1 -14442.499,E2 -14442.499} C_VEL
LIN {X 0,Y 333.597,Z 168.427,A -85,B 0,C 180,E1 -14445.954,E2 -14445.954} C_VEL
LIN {X 0,Y 333.605,Z 168.428,A -85,B 0,C 180,E1 -14449.325,E2 -14449.325} C_VEL
LIN {X 0,Y 333.662,Z 168.421,A -85,B 0,C 180,E1 -14453.169,E2 -14453.169} C_VEL
LIN {X 0,Y 333.673,Z 168.419,A -85,B 0,C 180,E1 -14455.34,E2 -14455.34} C_VEL
LIN {X 0,Y 333.622,Z 168.428,A -85,B 0,C 180,E1 -14458.22,E2 -14458.22} C_VEL
LIN {X 0,Y 333.696,Z 168.485,A -85,B 0,C 180,E1 -14460.031,E2 -14460.031} C_VEL
LIN {X 0,Y 335.625,Z 178.034,A -85,B 0,C 180,E1 -14462.906,E2 -14462.906} C_VEL
LIN {X 0,Y 337.259,Z 186.732,A -85,B 0,C 180,E1 -14465.368,E2 -14465.368} C_VEL
LIN {X 0,Y 337.268,Z 189.435,A -85,B 0,C 180,E1 -14466.089,E2 -14466.089} C_VEL
LIN {X 0,Y 336.964,Z 192.227,A -85,B 0,C 180,E1 -14466.72,E2 -14466.72} C_VEL
LIN {X 0,Y 342.46,Z 226.294,A -85,B 0,C 180,E1 -14467.893,E2 -14467.893} C_VEL
LIN {X 0,Y 340.883,Z 300.316,A -85,B 0,C 180,E1 -14469.561,E2 -14469.561} C_VEL
LIN {X 0,Y 340.189,Z 313.941,A -85,B 0,C 180,E1 -14470.108,E2 -14470.108} C_VEL
LIN {X 0,Y 339.201,Z 326.83,A -85,B 0,C 180,E1 -14470.874,E2 -14470.874} C_VEL
LIN {X 0,Y 338.134,Z 338.616,A -85,B 0,C 180,E1 -14471.833,E2 -14471.833} C_VEL
LIN {X 0,Y 336.987,Z 350.008,A -85,B 0,C 180,E1 -14473.023,E2 -14473.023} C_VEL
LIN {X 0,Y 335.985,Z 360.314,A -85,B 0,C 180,E1 -14474.379,E2 -14474.379} C_VEL
LIN {X 0,Y 334.836,Z 370.345,A -85,B 0,C 180,E1 -14476.031,E2 -14476.031} C_VEL
LIN {X 0,Y 333.722,Z 379.186,A -85,B 0,C 180,E1 -14477.842,E2 -14477.842} C_VEL
LIN {X 0,Y 333.002,Z 386.229,A -85,B 0,C 180,E1 -14479.665,E2 -14479.665} C_VEL
LIN {X 0,Y 332.481,Z 391.856,A -85,B 0,C 180,E1 -14481.49,E2 -14481.49} C_VEL
LIN {X 0,Y 332.16,Z 396.26,A -85,B 0,C 180,E1 -14483.316,E2 -14483.316} C_VEL
LIN {X 0,Y 331.97,Z 399.566,A -85,B 0,C 180,E1 -14485.141,E2 -14485.141} C_VEL
LIN {X 0,Y 331.955,Z 401.206,A -85,B 0,C 180,E1 -14486.357,E2 -14486.357} C_VEL
LIN {X 0,Y 331.886,Z 402.434,A -85,B 0,C 180,E1 -14487.571,E2 -14487.571} C_VEL
LIN {X 0,Y 331.867,Z 403.22,A -85,B 0,C 180,E1 -14488.785,E2 -14488.785} C_VEL
LIN {X 0,Y 331.9,Z 403.59,A -85,B 0,C 180,E1 -14489.999,E2 -14489.999} C_VEL
LIN {X 0,Y 331.866,Z 403.567,A -85,B 0,C 180,E1 -14491.212,E2 -14491.212} C_VEL
LIN {X 0,Y 331.886,Z 403.155,A -85,B 0,C 180,E1 -14492.426,E2 -14492.426} C_VEL
LIN {X 0,Y 331.966,Z 402.311,A -85,B 0,C 180,E1 -14493.64,E2 -14493.64} C_VEL
LIN {X 0,Y 332.088,Z 399.612,A -85,B 0,C 180,E1 -14495.917,E2 -14495.917} C_VEL
LIN {X 0,Y 332.427,Z 396.035,A -85,B 0,C 180,E1 -14497.897,E2 -14497.897} C_VEL
LIN {X 0,Y 332.936,Z 391.619,A -85,B 0,C 180,E1 -14499.721,E2 -14499.721} C_VEL
LIN {X 0,Y 333.707,Z 386.009,A -85,B 0,C 180,E1 -14501.54,E2 -14501.54} C_VEL
LIN {X 0,Y 334.739,Z 379.017,A -85,B 0,C 180,E1 -14503.351,E2 -14503.351} C_VEL
LIN {X 0,Y 336.135,Z 370.265,A -85,B 0,C 180,E1 -14505.149,E2 -14505.149} C_VEL
LIN {X 0,Y 337.095,Z 362.607,A -85,B 0,C 180,E1 -14506.454,E2 -14506.454} C_VEL
LIN {X 0,Y 338.453,Z 352.7,A -85,B 0,C 180,E1 -14507.834,E2 -14507.834} C_VEL
LIN {X 0,Y 339.78,Z 342.237,A -85,B 0,C 180,E1 -14509.011,E2 -14509.011} C_VEL
LIN {X 0,Y 341.208,Z 330.72,A -85,B 0,C 180,E1 -14510.023,E2 -14510.023} C_VEL
LIN {X 0,Y 342.411,Z 317.604,A -85,B 0,C 180,E1 -14510.891,E2 -14510.891} C_VEL
LIN {X 0,Y 343.371,Z 304.486,A -85,B 0,C 180,E1 -14511.498,E2 -14511.498} C_VEL
LIN {X 0,Y 343.901,Z 289.289,A -85,B 0,C 180,E1 -14511.921,E2 -14511.921} C_VEL
LIN {X 0,Y 345.535,Z 227.525,A -85,B 0,C 180,E1 -14513.308,E2 -14513.308} C_VEL
LIN {X 0,Y 341.96,Z 206.99,A -85,B 0,C 180,E1 -14514.13,E2 -14514.13} C_VEL
LIN {X 0,Y 338.559,Z 191.605,A -85,B 0,C 180,E1 -14514.845,E2 -14514.845} C_VEL
LIN {X 0,Y 338.3,Z 189.909,A -85,B 0,C 180,E1 -14515.204,E2 -14515.204} C_VEL
LIN {X 0,Y 336.701,Z 181.703,A -85,B 0,C 180,E1 -14517.639,E2 -14517.639} C_VEL
LIN {X 0,Y 334.611,Z 172.347,A -85,B 0,C 180,E1 -14520.554,E2 -14520.554} C_VEL
LIN {X 0,Y 333.673,Z 168.454,A -85,B 0,C 180,E1 -14521.911,E2 -14521.911} C_VEL
LIN {X 0,Y 333.68,Z 168.422,A -85,B 0,C 180,E1 -14524.772,E2 -14524.772} C_VEL
LIN {X 0,Y 333.637,Z 168.427,A -85,B 0,C 180,E1 -14527.651,E2 -14527.651} C_VEL
LIN {X 0,Y 333.597,Z 168.431,A -85,B 0,C 180,E1 -14530.772,E2 -14530.772} C_VEL
LIN {X 0,Y 333.583,Z 168.43,A -85,B 0,C 180,E1 -14534.248,E2 -14534.248} C_VEL
LIN {X 0,Y 333.628,Z 168.429,A -85,B 0,C 180,E1 -14537.616,E2 -14537.616} C_VEL
LIN {X 0,Y 333.626,Z 168.428,A -85,B 0,C 180,E1 -14541.205,E2 -14541.205} C_VEL
LIN {X 0,Y 333.665,Z 168.422,A -85,B 0,C 180,E1 -14543.859,E2 -14543.859} C_VEL
LIN {X 0,Y 333.635,Z 168.426,A -85,B 0,C 180,E1 -14547.412,E2 -14547.412} C_VEL
LIN {X 0,Y 333.64,Z 168.428,A -85,B 0,C 180,E1 -14551.021,E2 -14551.021} C_VEL
LIN {X 0,Y 333.684,Z 168.42,A -85,B 0,C 180,E1 -14555.087,E2 -14555.087} C_VEL
LIN {X 0,Y 333.653,Z 168.424,A -85,B 0,C 180,E1 -14559.017,E2 -14559.017} C_VEL
LIN {X 0,Y 333.73,Z 168.409,A -85,B 0,C 180,E1 -14561.585,E2 -14561.585} C_VEL
LIN {X 0,Y 333.797,Z 168.401,A -85,B 0,C 180,E1 -14565.576,E2 -14565.576} C_VEL
LIN {X 0,Y 333.805,Z 168.398,A -85,B 0,C 180,E1 -14569.077,E2 -14569.077} C_VEL
LIN {X 0,Y 333.959,Z 168.379,A -85,B 0,C 180,E1 -14572.746,E2 -14572.746} C_VEL
LIN {X 0,Y 333.778,Z 168.406,A -85,B 0,C 180,E1 -14575.168,E2 -14575.168} C_VEL
LIN {X 0,Y 334.058,Z 168.37,A -85,B 0,C 180,E1 -14577.588,E2 -14577.588} C_VEL
LIN {X 0,Y 334.067,Z 168.372,A -85,B 0,C 180,E1 -14581.205,E2 -14581.205} C_VEL
LIN {X 0,Y 333.793,Z 168.4,A -85,B 0,C 180,E1 -14583.621,E2 -14583.621} C_VEL
LIN {X 0,Y 333.962,Z 168.382,A -85,B 0,C 180,E1 -14586.693,E2 -14586.693} C_VEL
LIN {X 0,Y 333.805,Z 168.402,A -85,B 0,C 180,E1 -14589.696,E2 -14589.696} C_VEL
LIN {X 0,Y 333.782,Z 168.407,A -85,B 0,C 180,E1 -14593.391,E2 -14593.391} C_VEL
LIN {X 0,Y 333.706,Z 168.418,A -85,B 0,C 180,E1 -14597.148,E2 -14597.148} C_VEL
LIN {X 0,Y 333.658,Z 168.423,A -85,B 0,C 180,E1 -14599.695,E2 -14599.695} C_VEL
LIN {X 0,Y 333.634,Z 168.427,A -85,B 0,C 180,E1 -14603.592,E2 -14603.592} C_VEL
LIN {X 0,Y 333.68,Z 168.545,A -85,B 0,C 180,E1 -14604.58,E2 -14604.58} C_VEL
LIN {X 0,Y 335.904,Z 178.188,A -85,B 0,C 180,E1 -14607.744,E2 -14607.744} C_VEL
LIN {X 0,Y 336.931,Z 182.505,A -85,B 0,C 180,E1 -14609.009,E2 -14609.009} C_VEL
LIN {X 0,Y 339.984,Z 189.75,A -85,B 0,C 180,E1 -14609.53,E2 -14609.53} C_VEL
LIN {X 0,Y 342.164,Z 195.583,A -85,B 0,C 180,E1 -14609.873,E2 -14609.873} C_VEL
LIN {X 0,Y 345.468,Z 211.823,A -85,B 0,C 180,E1 -14610.569,E2 -14610.569} C_VEL
LIN {X 0,Y 345.808,Z 215.595,A -85,B 0,C 180,E1 -14610.692,E2 -14610.692} C_VEL
LIN {X 0,Y 343.727,Z 290.461,A -85,B 0,C 180,E1 -14612.403,E2 -14612.403} C_VEL
LIN {X 0,Y 342.957,Z 303.487,A -85,B 0,C 180,E1 -14612.923,E2 -14612.923} C_VEL
LIN {X 0,Y 341.98,Z 316.549,A -85,B 0,C 180,E1 -14613.701,E2 -14613.701} C_VEL
LIN {X 0,Y 340.856,Z 327.774,A -85,B 0,C 180,E1 -14614.604,E2 -14614.604} C_VEL
LIN {X 0,Y 339.521,Z 338.741,A -85,B 0,C 180,E1 -14615.726,E2 -14615.726} C_VEL
LIN {X 0,Y 338.076,Z 349.262,A -85,B 0,C 180,E1 -14617.074,E2 -14617.074} C_VEL
LIN {X 0,Y 336.706,Z 358.728,A -85,B 0,C 180,E1 -14618.589,E2 -14618.589} C_VEL
LIN {X 0,Y 335.402,Z 367.34,A -85,B 0,C 180,E1 -14620.305,E2 -14620.305} C_VEL
LIN {X 0,Y 334.149,Z 375.343,A -85,B 0,C 180,E1 -14622.301,E2 -14622.301} C_VEL
LIN {X 0,Y 333.302,Z 381.262,A -85,B 0,C 180,E1 -14624.202,E2 -14624.202} C_VEL
LIN {X 0,Y 332.761,Z 385.435,A -85,B 0,C 180,E1 -14625.896,E2 -14625.896} C_VEL
LIN {X 0,Y 332.338,Z 388.904,A -85,B 0,C 180,E1 -14627.743,E2 -14627.743} C_VEL
LIN {X 0,Y 331.944,Z 391.419,A -85,B 0,C 180,E1 -14629.658,E2 -14629.658} C_VEL
LIN {X 0,Y 331.705,Z 392.921,A -85,B 0,C 180,E1 -14631.622,E2 -14631.622} C_VEL
LIN {X 0,Y 331.646,Z 393.36,A -85,B 0,C 180,E1 -14633.635,E2 -14633.635} C_VEL
LIN {X 0,Y 331.643,Z 392.632,A -85,B 0,C 180,E1 -14635.736,E2 -14635.736} C_VEL
LIN {X 0,Y 331.87,Z 390.446,A -85,B 0,C 180,E1 -14638.035,E2 -14638.035} C_VEL
LIN {X 0,Y 332.193,Z 387.079,A -85,B 0,C 180,E1 -14640.158,E2 -14640.158} C_VEL
LIN {X 0,Y 332.648,Z 382.167,A -85,B 0,C 180,E1 -14642.304,E2 -14642.304} C_VEL
LIN {X 0,Y 333.251,Z 375.854,A -85,B 0,C 180,E1 -14644.383,E2 -14644.383} C_VEL
LIN {X 0,Y 333.997,Z 369.215,A -85,B 0,C 180,E1 -14646.107,E2 -14646.107} C_VEL
LIN {X 0,Y 334.909,Z 361.093,A -85,B 0,C 180,E1 -14647.809,E2 -14647.809} C_VEL
LIN {X 0,Y 336.077,Z 351.615,A -85,B 0,C 180,E1 -14649.407,E2 -14649.407} C_VEL
LIN {X 0,Y 337.228,Z 341.099,A -85,B 0,C 180,E1 -14650.84,E2 -14650.84} C_VEL
LIN {X 0,Y 338.343,Z 329.868,A -85,B 0,C 180,E1 -14652.048,E2 -14652.048} C_VEL
LIN {X 0,Y 339.377,Z 317.866,A -85,B 0,C 180,E1 -14653.055,E2 -14653.055} C_VEL
LIN {X 0,Y 340.08,Z 306.195,A -85,B 0,C 180,E1 -14653.802,E2 -14653.802} C_VEL
LIN {X 0,Y 340.801,Z 293.189,A -85,B 0,C 180,E1 -14654.374,E2 -14654.374} C_VEL
LIN {X 0,Y 341.329,Z 275.6,A -85,B 0,C 180,E1 -14654.824,E2 -14654.824} C_VEL
LIN {X 0,Y 342.576,Z 211.59,A -85,B 0,C 180,E1 -14656.242,E2 -14656.242} C_VEL
LIN {X 0,Y 337.769,Z 186.3,A -85,B 0,C 180,E1 -14657.13,E2 -14657.13} C_VEL
LIN {X 0,Y 336.431,Z 182.225,A -85,B 0,C 180,E1 -14657.37,E2 -14657.37} C_VEL
LIN {X 0,Y 334.606,Z 172.213,A -85,B 0,C 180,E1 -14660.328,E2 -14660.328} C_VEL
LIN {X 0,Y 333.942,Z 168.435,A -85,B 0,C 180,E1 -14661.573,E2 -14661.573} C_VEL
LIN {X 0,Y 334.013,Z 168.381,A -85,B 0,C 180,E1 -14663.962,E2 -14663.962} C_VEL
LIN {X 0,Y 334.102,Z 168.369,A -85,B 0,C 180,E1 -14667.59,E2 -14667.59} C_VEL
LIN {X 0,Y 334.243,Z 168.35,A -85,B 0,C 180,E1 -14670.001,E2 -14670.001} C_VEL
LIN {X 0,Y 334.103,Z 168.365,A -85,B 0,C 180,E1 -14672.412,E2 -14672.412} C_VEL
LIN {X 0,Y 334.006,Z 168.379,A -85,B 0,C 180,E1 -14676.04,E2 -14676.04} C_VEL
LIN {X 0,Y 333.819,Z 168.404,A -85,B 0,C 180,E1 -14679.697,E2 -14679.697} C_VEL
LIN {X 0,Y 333.795,Z 168.407,A -85,B 0,C 180,E1 -14683.393,E2 -14683.393} C_VEL
LIN {X 0,Y 333.746,Z 168.413,A -85,B 0,C 180,E1 -14687.147,E2 -14687.147} C_VEL
LIN {X 0,Y 333.737,Z 168.412,A -85,B 0,C 180,E1 -14689.691,E2 -14689.691} C_VEL
LIN {X 0,Y 333.692,Z 168.416,A -85,B 0,C 180,E1 -14692.279,E2 -14692.279} C_VEL
LIN {X 0,Y 333.735,Z 168.409,A -85,B 0,C 180,E1 -14696.247,E2 -14696.247} C_VEL
LIN {X 0,Y 333.687,Z 168.419,A -85,B 0,C 180,E1 -14698.891,E2 -14698.891} C_VEL
LIN {X 0,Y 333.044,Z 168.506,A -85,B 0,C 180,E1 -14699.898,E2 -14699.898} C_VEL
LIN {X 0,Y 330.188,Z 168.862,A -85,B 0,C 180,E1 -14701.535,E2 -14701.535} C_VEL
LIN {X 0,Y 327.746,Z 169.161,A -85,B 0,C 180,E1 -14702.862,E2 -14702.862} C_VEL
LIN {X 0,Y 326.689,Z 169.287,A -85,B 0,C 180,E1 -14703.889,E2 -14703.889} C_VEL
LIN {X 0,Y 326.599,Z 169.297,A -85,B 0,C 180,E1 -14704.238,E2 -14704.238} C_VEL
LIN {X 0,Y 326.627,Z 169.296,A -85,B 0,C 180,E1 -14707.239,E2 -14707.239} C_VEL
LIN {X 0,Y 326.578,Z 169.305,A -85,B 0,C 180,E1 -14711.132,E2 -14711.132} C_VEL
LIN {X 0,Y 326.556,Z 169.309,A -85,B 0,C 180,E1 -14714.749,E2 -14714.749} C_VEL
LIN {X 0,Y 326.574,Z 169.299,A -85,B 0,C 180,E1 -14718.155,E2 -14718.155} C_VEL
LIN {X 0,Y 326.586,Z 169.299,A -85,B 0,C 180,E1 -14721.387,E2 -14721.387} C_VEL
LIN {X 0,Y 326.62,Z 169.3,A -85,B 0,C 180,E1 -14724.852,E2 -14724.852} C_VEL
LIN {X 0,Y 326.608,Z 169.298,A -85,B 0,C 180,E1 -14727.456,E2 -14727.456} C_VEL
LIN {X 0,Y 326.617,Z 169.301,A -85,B 0,C 180,E1 -14730.337,E2 -14730.337} C_VEL
LIN {X 0,Y 326.644,Z 169.296,A -85,B 0,C 180,E1 -14734.645,E2 -14734.645} C_VEL
LIN {X 0,Y 326.622,Z 169.299,A -85,B 0,C 180,E1 -14738.544,E2 -14738.544} C_VEL
LIN {X 0,Y 326.746,Z 169.281,A -85,B 0,C 180,E1 -14741.178,E2 -14741.178} C_VEL
LIN {X 0,Y 326.765,Z 169.278,A -85,B 0,C 180,E1 -14745.434,E2 -14745.434} C_VEL
LIN {X 0,Y 326.759,Z 169.279,A -85,B 0,C 180,E1 -14748.839,E2 -14748.839} C_VEL
LIN {X 0,Y 326.914,Z 169.26,A -85,B 0,C 180,E1 -14752.589,E2 -14752.589} C_VEL
LIN {X 0,Y 326.748,Z 169.281,A -85,B 0,C 180,E1 -14755.065,E2 -14755.065} C_VEL
LIN {X 0,Y 327.01,Z 169.251,A -85,B 0,C 180,E1 -14757.537,E2 -14757.537} C_VEL
LIN {X 0,Y 327.03,Z 169.244,A -85,B 0,C 180,E1 -14761.232,E2 -14761.232} C_VEL
LIN {X 0,Y 326.761,Z 169.279,A -85,B 0,C 180,E1 -14763.7,E2 -14763.7} C_VEL
LIN {X 0,Y 326.941,Z 169.257,A -85,B 0,C 180,E1 -14766.171,E2 -14766.171} C_VEL
LIN {X 0,Y 326.785,Z 169.279,A -85,B 0,C 180,E1 -14769.908,E2 -14769.908} C_VEL
LIN {X 0,Y 326.759,Z 169.28,A -85,B 0,C 180,E1 -14773.686,E2 -14773.686} C_VEL
LIN {X 0,Y 326.657,Z 169.295,A -85,B 0,C 180,E1 -14777.531,E2 -14777.531} C_VEL
LIN {X 0,Y 326.613,Z 169.302,A -85,B 0,C 180,E1 -14781.458,E2 -14781.458} C_VEL
LIN {X 0,Y 326.603,Z 169.299,A -85,B 0,C 180,E1 -14785.492,E2 -14785.492} C_VEL
LIN {X 0,Y 326.616,Z 169.299,A -85,B 0,C 180,E1 -14789.664,E2 -14789.664} C_VEL
LIN {X 0,Y 326.616,Z 169.301,A -85,B 0,C 180,E1 -14792.945,E2 -14792.945} C_VEL
LIN {X 0,Y 326.613,Z 169.299,A -85,B 0,C 180,E1 -14795.52,E2 -14795.52} C_VEL
LIN {X 0,Y 326.591,Z 169.302,A -85,B 0,C 180,E1 -14799.222,E2 -14799.222} C_VEL
LIN {X 0,Y 326.575,Z 169.307,A -85,B 0,C 180,E1 -14802.971,E2 -14802.971} C_VEL
LIN {X 0,Y 326.575,Z 169.306,A -85,B 0,C 180,E1 -14807.029,E2 -14807.029} C_VEL
LIN {X 0,Y 326.589,Z 169.305,A -85,B 0,C 180,E1 -14810.778,E2 -14810.778} C_VEL
LIN {X 0,Y 326.611,Z 169.303,A -85,B 0,C 180,E1 -14814.479,E2 -14814.479} C_VEL
LIN {X 0,Y 326.604,Z 169.3,A -85,B 0,C 180,E1 -14817.454,E2 -14817.454} C_VEL
LIN {X 0,Y 326.637,Z 169.427,A -85,B 0,C 180,E1 -14819.729,E2 -14819.729} C_VEL
LIN {X 0,Y 328.82,Z 180.127,A -85,B 0,C 180,E1 -14822.987,E2 -14822.987} C_VEL
LIN {X 0,Y 330.393,Z 188.816,A -85,B 0,C 180,E1 -14825.492,E2 -14825.492} C_VEL
LIN {X 0,Y 330.138,Z 191.89,A -85,B 0,C 180,E1 -14826.262,E2 -14826.262} C_VEL
LIN {X 0,Y 332.213,Z 204.668,A -85,B 0,C 180,E1 -14826.752,E2 -14826.752} C_VEL
LIN {X 0,Y 335.835,Z 228.276,A -85,B 0,C 180,E1 -14827.547,E2 -14827.547} C_VEL
LIN {X 0,Y 334.117,Z 300.51,A -85,B 0,C 180,E1 -14829.208,E2 -14829.208} C_VEL
LIN {X 0,Y 333.372,Z 314.025,A -85,B 0,C 180,E1 -14829.764,E2 -14829.764} C_VEL
LIN {X 0,Y 332.377,Z 326.85,A -85,B 0,C 180,E1 -14830.546,E2 -14830.546} C_VEL
LIN {X 0,Y 331.19,Z 339.406,A -85,B 0,C 180,E1 -14831.599,E2 -14831.599} C_VEL
LIN {X 0,Y 330.031,Z 350.641,A -85,B 0,C 180,E1 -14832.813,E2 -14832.813} C_VEL
LIN {X 0,Y 329.01,Z 360.657,A -85,B 0,C 180,E1 -14834.179,E2 -14834.179} C_VEL
LIN {X 0,Y 327.891,Z 369.891,A -85,B 0,C 180,E1 -14835.729,E2 -14835.729} C_VEL
LIN {X 0,Y 326.763,Z 378.802,A -85,B 0,C 180,E1 -14837.579,E2 -14837.579} C_VEL
LIN {X 0,Y 325.98,Z 385.914,A -85,B 0,C 180,E1 -14839.439,E2 -14839.439} C_VEL
LIN {X 0,Y 325.419,Z 391.584,A -85,B 0,C 180,E1 -14841.304,E2 -14841.304} C_VEL
LIN {X 0,Y 325.077,Z 396.028,A -85,B 0,C 180,E1 -14843.17,E2 -14843.17} C_VEL
LIN {X 0,Y 324.887,Z 399.369,A -85,B 0,C 180,E1 -14845.035,E2 -14845.035} C_VEL
LIN {X 0,Y 324.863,Z 401.025,A -85,B 0,C 180,E1 -14846.278,E2 -14846.278} C_VEL
LIN {X 0,Y 324.807,Z 402.269,A -85,B 0,C 180,E1 -14847.518,E2 -14847.518} C_VEL
LIN {X 0,Y 324.779,Z 403.086,A -85,B 0,C 180,E1 -14848.759,E2 -14848.759} C_VEL
LIN {X 0,Y 324.808,Z 403.471,A -85,B 0,C 180,E1 -14849.999,E2 -14849.999} C_VEL
LIN {X 0,Y 324.808,Z 403.067,A -85,B 0,C 180,E1 -14852.479,E2 -14852.479} C_VEL
LIN {X 0,Y 324.876,Z 402.257,A -85,B 0,C 180,E1 -14853.72,E2 -14853.72} C_VEL
LIN {X 0,Y 324.999,Z 399.837,A -85,B 0,C 180,E1 -14855.878,E2 -14855.878} C_VEL
LIN {X 0,Y 325.39,Z 396.048,A -85,B 0,C 180,E1 -14858.069,E2 -14858.069} C_VEL
LIN {X 0,Y 325.908,Z 391.666,A -85,B 0,C 180,E1 -14859.933,E2 -14859.933} C_VEL
LIN {X 0,Y 326.704,Z 386.094,A -85,B 0,C 180,E1 -14861.791,E2 -14861.791} C_VEL
LIN {X 0,Y 327.833,Z 379.148,A -85,B 0,C 180,E1 -14863.638,E2 -14863.638} C_VEL
LIN {X 0,Y 329.283,Z 370.462,A -85,B 0,C 180,E1 -14865.472,E2 -14865.472} C_VEL
LIN {X 0,Y 330.511,Z 361.586,A -85,B 0,C 180,E1 -14867,E2 -14867} C_VEL
LIN {X 0,Y 331.911,Z 351.894,A -85,B 0,C 180,E1 -14868.357,E2 -14868.357} C_VEL
LIN {X 0,Y 333.279,Z 341.311,A -85,B 0,C 180,E1 -14869.556,E2 -14869.556} C_VEL
LIN {X 0,Y 334.776,Z 329.519,A -85,B 0,C 180,E1 -14870.586,E2 -14870.586} C_VEL
LIN {X 0,Y 336.055,Z 316.109,A -85,B 0,C 180,E1 -14871.466,E2 -14871.466} C_VEL
LIN {X 0,Y 337.026,Z 303.143,A -85,B 0,C 180,E1 -14872.044,E2 -14872.044} C_VEL
LIN {X 0,Y 337.507,Z 288.719,A -85,B 0,C 180,E1 -14872.444,E2 -14872.444} C_VEL
LIN {X 0,Y 339.13,Z 227.894,A -85,B 0,C 180,E1 -14873.843,E2 -14873.843} C_VEL
LIN {X 0,Y 335.461,Z 207.116,A -85,B 0,C 180,E1 -14874.707,E2 -14874.707} C_VEL
LIN {X 0,Y 332.449,Z 194.015,A -85,B 0,C 180,E1 -14875.343,E2 -14875.343} C_VEL
LIN {X 0,Y 331.408,Z 191.057,A -85,B 0,C 180,E1 -14875.572,E2 -14875.572} C_VEL
LIN {X 0,Y 329.547,Z 181.958,A -85,B 0,C 180,E1 -14878.303,E2 -14878.303} C_VEL
LIN {X 0,Y 327.364,Z 172.439,A -85,B 0,C 180,E1 -14881.371,E2 -14881.371} C_VEL
LIN {X 0,Y 326.607,Z 169.335,A -85,B 0,C 180,E1 -14882.52,E2 -14882.52} C_VEL
LIN {X 0,Y 326.606,Z 169.303,A -85,B 0,C 180,E1 -14885.518,E2 -14885.518} C_VEL
LIN {X 0,Y 326.581,Z 169.307,A -85,B 0,C 180,E1 -14889.22,E2 -14889.22} C_VEL
LIN {X 0,Y 326.565,Z 169.309,A -85,B 0,C 180,E1 -14892.969,E2 -14892.969} C_VEL
LIN {X 0,Y 326.564,Z 169.305,A -85,B 0,C 180,E1 -14897.027,E2 -14897.027} C_VEL
LIN {X 0,Y 326.574,Z 169.304,A -85,B 0,C 180,E1 -14901.384,E2 -14901.384} C_VEL
LIN {X 0,Y 326.609,Z 169.299,A -85,B 0,C 180,E1 -14904.85,E2 -14904.85} C_VEL
LIN {X 0,Y 326.599,Z 169.302,A -85,B 0,C 180,E1 -14907.454,E2 -14907.454} C_VEL
LIN {X 0,Y 326.605,Z 169.299,A -85,B 0,C 180,E1 -14910.335,E2 -14910.335} C_VEL
LIN {X 0,Y 326.631,Z 169.299,A -85,B 0,C 180,E1 -14914.644,E2 -14914.644} C_VEL
LIN {X 0,Y 326.604,Z 169.301,A -85,B 0,C 180,E1 -14918.542,E2 -14918.542} C_VEL
LIN {X 0,Y 326.653,Z 169.293,A -85,B 0,C 180,E1 -14922.469,E2 -14922.469} C_VEL
LIN {X 0,Y 326.748,Z 169.281,A -85,B 0,C 180,E1 -14926.314,E2 -14926.314} C_VEL
LIN {X 0,Y 326.771,Z 169.278,A -85,B 0,C 180,E1 -14930.092,E2 -14930.092} C_VEL
LIN {X 0,Y 326.941,Z 169.256,A -85,B 0,C 180,E1 -14933.829,E2 -14933.829} C_VEL
LIN {X 0,Y 327.001,Z 169.25,A -85,B 0,C 180,E1 -14937.536,E2 -14937.536} C_VEL
LIN {X 0,Y 327.034,Z 169.248,A -85,B 0,C 180,E1 -14941.231,E2 -14941.231} C_VEL
LIN {X 0,Y 326.742,Z 169.278,A -85,B 0,C 180,E1 -14943.699,E2 -14943.699} C_VEL
LIN {X 0,Y 326.918,Z 169.258,A -85,B 0,C 180,E1 -14946.688,E2 -14946.688} C_VEL
LIN {X 0,Y 326.768,Z 169.28,A -85,B 0,C 180,E1 -14949.907,E2 -14949.907} C_VEL
LIN {X 0,Y 326.745,Z 169.283,A -85,B 0,C 180,E1 -14953.685,E2 -14953.685} C_VEL
LIN {X 0,Y 326.651,Z 169.296,A -85,B 0,C 180,E1 -14957.53,E2 -14957.53} C_VEL
LIN {X 0,Y 326.601,Z 169.303,A -85,B 0,C 180,E1 -14961.457,E2 -14961.457} C_VEL
LIN {X 0,Y 326.635,Z 169.405,A -85,B 0,C 180,E1 -14963.961,E2 -14963.961} C_VEL
LIN {X 0,Y 328.741,Z 178.383,A -85,B 0,C 180,E1 -14967.019,E2 -14967.019} C_VEL
LIN {X 0,Y 329.743,Z 182.699,A -85,B 0,C 180,E1 -14968.316,E2 -14968.316} C_VEL
LIN {X 0,Y 334.345,Z 193.262,A -85,B 0,C 180,E1 -14969.098,E2 -14969.098} C_VEL
LIN {X 0,Y 336.324,Z 198.756,A -85,B 0,C 180,E1 -14969.43,E2 -14969.43} C_VEL
LIN {X 0,Y 339.501,Z 214.896,A -85,B 0,C 180,E1 -14970.132,E2 -14970.132} C_VEL
LIN {X 0,Y 337.308,Z 290.797,A -85,B 0,C 180,E1 -14971.904,E2 -14971.904} C_VEL
LIN {X 0,Y 336.505,Z 303.765,A -85,B 0,C 180,E1 -14972.434,E2 -14972.434} C_VEL
LIN {X 0,Y 335.492,Z 316.678,A -85,B 0,C 180,E1 -14973.218,E2 -14973.218} C_VEL
LIN {X 0,Y 334.166,Z 328.923,A -85,B 0,C 180,E1 -14974.233,E2 -14974.233} C_VEL
LIN {X 0,Y 332.826,Z 339.496,A -85,B 0,C 180,E1 -14975.356,E2 -14975.356} C_VEL
LIN {X 0,Y 331.248,Z 350.33,A -85,B 0,C 180,E1 -14976.794,E2 -14976.794} C_VEL
LIN {X 0,Y 329.981,Z 358.535,A -85,B 0,C 180,E1 -14978.144,E2 -14978.144} C_VEL
LIN {X 0,Y 328.587,Z 367.29,A -85,B 0,C 180,E1 -14979.915,E2 -14979.915} C_VEL
LIN {X 0,Y 327.442,Z 374.445,A -85,B 0,C 180,E1 -14981.709,E2 -14981.709} C_VEL
LIN {X 0,Y 326.494,Z 380.287,A -85,B 0,C 180,E1 -14983.536,E2 -14983.536} C_VEL
LIN {X 0,Y 325.83,Z 384.935,A -85,B 0,C 180,E1 -14985.38,E2 -14985.38} C_VEL
LIN {X 0,Y 325.334,Z 388.553,A -85,B 0,C 180,E1 -14987.263,E2 -14987.263} C_VEL
LIN {X 0,Y 324.872,Z 391.569,A -85,B 0,C 180,E1 -14989.537,E2 -14989.537} C_VEL
LIN {X 0,Y 324.641,Z 392.863,A -85,B 0,C 180,E1 -14991.2,E2 -14991.2} C_VEL
LIN {X 0,Y 324.537,Z 393.476,A -85,B 0,C 180,E1 -14993.249,E2 -14993.249} C_VEL
LIN {X 0,Y 324.554,Z 392.958,A -85,B 0,C 180,E1 -14995.371,E2 -14995.371} C_VEL
LIN {X 0,Y 324.706,Z 391.133,A -85,B 0,C 180,E1 -14997.577,E2 -14997.577} C_VEL
LIN {X 0,Y 325.074,Z 387.841,A -85,B 0,C 180,E1 -14999.857,E2 -14999.857} C_VEL
LIN {X 0,Y 325.4,Z 384.212,A -85,B 0,C 180,E1 -15001.632,E2 -15001.632} C_VEL
LIN {X 0,Y 326.011,Z 378.454,A -85,B 0,C 180,E1 -15003.775,E2 -15003.775} C_VEL
LIN {X 0,Y 326.698,Z 372.119,A -85,B 0,C 180,E1 -15005.608,E2 -15005.608} C_VEL
LIN {X 0,Y 327.544,Z 364.8,A -85,B 0,C 180,E1 -15007.313,E2 -15007.313} C_VEL
LIN {X 0,Y 328.649,Z 355.823,A -85,B 0,C 180,E1 -15009.006,E2 -15009.006} C_VEL
LIN {X 0,Y 329.835,Z 345.657,A -85,B 0,C 180,E1 -15010.555,E2 -15010.555} C_VEL
LIN {X 0,Y 331.013,Z 334.904,A -85,B 0,C 180,E1 -15011.856,E2 -15011.856} C_VEL
LIN {X 0,Y 332.048,Z 323.818,A -85,B 0,C 180,E1 -15012.924,E2 -15012.924} C_VEL
LIN {X 0,Y 332.985,Z 311.499,A -85,B 0,C 180,E1 -15013.841,E2 -15013.841} C_VEL
LIN {X 0,Y 333.794,Z 298.255,A -85,B 0,C 180,E1 -15014.538,E2 -15014.538} C_VEL
LIN {X 0,Y 334.363,Z 284.813,A -85,B 0,C 180,E1 -15014.985,E2 -15014.985} C_VEL
LIN {X 0,Y 335.947,Z 212.979,A -85,B 0,C 180,E1 -15016.611,E2 -15016.611} C_VEL
LIN {X 0,Y 331.439,Z 188.726,A -85,B 0,C 180,E1 -15017.48,E2 -15017.48} C_VEL
LIN {X 0,Y 329.367,Z 182.555,A -85,B 0,C 180,E1 -15017.798,E2 -15017.798} C_VEL
LIN {X 0,Y 328.242,Z 176.672,A -85,B 0,C 180,E1 -15019.516,E2 -15019.516} C_VEL
LIN {X 0,Y 326.913,Z 169.312,A -85,B 0,C 180,E1 -15021.902,E2 -15021.902} C_VEL
LIN {X 0,Y 326.987,Z 169.257,A -85,B 0,C 180,E1 -15023.832,E2 -15023.832} C_VEL
LIN {X 0,Y 327.043,Z 169.248,A -85,B 0,C 180,E1 -15027.538,E2 -15027.538} C_VEL
LIN {X 0,Y 327.194,Z 169.228,A -85,B 0,C 180,E1 -15030.001,E2 -15030.001} C_VEL
LIN {X 0,Y 327.043,Z 169.245,A -85,B 0,C 180,E1 -15032.465,E2 -15032.465} C_VEL
LIN {X 0,Y 326.98,Z 169.253,A -85,B 0,C 180,E1 -15036.171,E2 -15036.171} C_VEL
LIN {X 0,Y 326.782,Z 169.279,A -85,B 0,C 180,E1 -15039.908,E2 -15039.908} C_VEL
LIN {X 0,Y 326.758,Z 169.283,A -85,B 0,C 180,E1 -15043.687,E2 -15043.687} C_VEL
LIN {X 0,Y 326.698,Z 169.29,A -85,B 0,C 180,E1 -15047.529,E2 -15047.529} C_VEL
LIN {X 0,Y 326.664,Z 169.291,A -85,B 0,C 180,E1 -15050.136,E2 -15050.136} C_VEL
LIN {X 0,Y 326.651,Z 169.292,A -85,B 0,C 180,E1 -15054.13,E2 -15054.13} C_VEL
LIN {X 0,Y 326.682,Z 169.289,A -85,B 0,C 180,E1 -15056.859,E2 -15056.859} C_VEL
LIN {X 0,Y 326.634,Z 169.297,A -85,B 0,C 180,E1 -15060.611,E2 -15060.611} C_VEL
LIN {X 0,Y 326.599,Z 169.297,A -85,B 0,C 180,E1 -15064.238,E2 -15064.238} C_VEL
LIN {X 0,Y 325.938,Z 169.382,A -85,B 0,C 180,E1 -15065.267,E2 -15065.267} C_VEL
LIN {X 0,Y 323.136,Z 169.734,A -85,B 0,C 180,E1 -15066.944,E2 -15066.944} C_VEL
LIN {X 0,Y 320.737,Z 170.035,A -85,B 0,C 180,E1 -15068.302,E2 -15068.302} C_VEL
LIN {X 0,Y 319.665,Z 170.165,A -85,B 0,C 180,E1 -15069.353,E2 -15069.353} C_VEL
LIN {X 0,Y 319.555,Z 170.176,A -85,B 0,C 180,E1 -15069.709,E2 -15069.709} C_VEL
LIN {X 0,Y 319.558,Z 170.177,A -85,B 0,C 180,E1 -15073.468,E2 -15073.468} C_VEL
LIN {X 0,Y 319.559,Z 170.173,A -85,B 0,C 180,E1 -15077.018,E2 -15077.018} C_VEL
LIN {X 0,Y 319.545,Z 170.176,A -85,B 0,C 180,E1 -15080.371,E2 -15080.371} C_VEL
LIN {X 0,Y 319.58,Z 170.178,A -85,B 0,C 180,E1 -15084.458,E2 -15084.458} C_VEL
LIN {X 0,Y 319.524,Z 170.182,A -85,B 0,C 180,E1 -15088.138,E2 -15088.138} C_VEL
LIN {X 0,Y 319.572,Z 170.175,A -85,B 0,C 180,E1 -15091.604,E2 -15091.604} C_VEL
LIN {X 0,Y 319.577,Z 170.173,A -85,B 0,C 180,E1 -15095.302,E2 -15095.302} C_VEL
LIN {X 0,Y 319.604,Z 170.17,A -85,B 0,C 180,E1 -15099.401,E2 -15099.401} C_VEL
LIN {X 0,Y 319.66,Z 170.168,A -85,B 0,C 180,E1 -15102.074,E2 -15102.074} C_VEL
LIN {X 0,Y 319.734,Z 170.157,A -85,B 0,C 180,E1 -15106.008,E2 -15106.008} C_VEL
LIN {X 0,Y 319.737,Z 170.158,A -85,B 0,C 180,E1 -15109.873,E2 -15109.873} C_VEL
LIN {X 0,Y 319.901,Z 170.136,A -85,B 0,C 180,E1 -15113.694,E2 -15113.694} C_VEL
LIN {X 0,Y 319.956,Z 170.129,A -85,B 0,C 180,E1 -15117.483,E2 -15117.483} C_VEL
LIN {X 0,Y 320,Z 170.12,A -85,B 0,C 180,E1 -15121.259,E2 -15121.259} C_VEL
LIN {X 0,Y 319.71,Z 170.155,A -85,B 0,C 180,E1 -15123.782,E2 -15123.782} C_VEL
LIN {X 0,Y 319.898,Z 170.133,A -85,B 0,C 180,E1 -15126.307,E2 -15126.307} C_VEL
LIN {X 0,Y 319.737,Z 170.155,A -85,B 0,C 180,E1 -15130.128,E2 -15130.128} C_VEL
LIN {X 0,Y 319.733,Z 170.152,A -85,B 0,C 180,E1 -15133.993,E2 -15133.993} C_VEL
LIN {X 0,Y 319.61,Z 170.17,A -85,B 0,C 180,E1 -15137.93,E2 -15137.93} C_VEL
LIN {X 0,Y 319.566,Z 170.176,A -85,B 0,C 180,E1 -15141.955,E2 -15141.955} C_VEL
LIN {X 0,Y 319.552,Z 170.173,A -85,B 0,C 180,E1 -15146.096,E2 -15146.096} C_VEL
LIN {X 0,Y 319.543,Z 170.181,A -85,B 0,C 180,E1 -15148.939,E2 -15148.939} C_VEL
LIN {X 0,Y 319.522,Z 170.181,A -85,B 0,C 180,E1 -15151.864,E2 -15151.864} C_VEL
LIN {X 0,Y 319.581,Z 170.175,A -85,B 0,C 180,E1 -15155.542,E2 -15155.542} C_VEL
LIN {X 0,Y 319.532,Z 170.178,A -85,B 0,C 180,E1 -15159.662,E2 -15159.662} C_VEL
LIN {X 0,Y 319.522,Z 170.182,A -85,B 0,C 180,E1 -15163.46,E2 -15163.46} C_VEL
LIN {X 0,Y 319.554,Z 170.18,A -85,B 0,C 180,E1 -15167.015,E2 -15167.015} C_VEL
LIN {X 0,Y 319.534,Z 170.183,A -85,B 0,C 180,E1 -15170.368,E2 -15170.368} C_VEL
LIN {X 0,Y 319.579,Z 170.179,A -85,B 0,C 180,E1 -15174.458,E2 -15174.458} C_VEL
LIN {X 0,Y 319.521,Z 170.185,A -85,B 0,C 180,E1 -15178.136,E2 -15178.136} C_VEL
LIN {X 0,Y 319.584,Z 170.248,A -85,B 0,C 180,E1 -15179.343,E2 -15179.343} C_VEL
LIN {X 0,Y 321.523,Z 179.695,A -85,B 0,C 180,E1 -15182.322,E2 -15182.322} C_VEL
LIN {X 0,Y 323.37,Z 189.65,A -85,B 0,C 180,E1 -15185.267,E2 -15185.267} C_VEL
LIN {X 0,Y 323.344,Z 191.845,A -85,B 0,C 180,E1 -15185.815,E2 -15185.815} C_VEL
LIN {X 0,Y 327.768,Z 219.674,A -85,B 0,C 180,E1 -15186.842,E2 -15186.842} C_VEL
LIN {X 0,Y 329.101,Z 229.45,A -85,B 0,C 180,E1 -15187.167,E2 -15187.167} C_VEL
LIN {X 0,Y 327.353,Z 300.567,A -85,B 0,C 180,E1 -15188.84,E2 -15188.84} C_VEL
LIN {X 0,Y 326.586,Z 314.02,A -85,B 0,C 180,E1 -15189.407,E2 -15189.407} C_VEL
LIN {X 0,Y 325.568,Z 326.809,A -85,B 0,C 180,E1 -15190.205,E2 -15190.205} C_VEL
LIN {X 0,Y 324.448,Z 338.559,A -85,B 0,C 180,E1 -15191.202,E2 -15191.202} C_VEL
LIN {X 0,Y 323.204,Z 349.925,A -85,B 0,C 180,E1 -15192.439,E2 -15192.439} C_VEL
LIN {X 0,Y 322.185,Z 359.214,A -85,B 0,C 180,E1 -15193.7,E2 -15193.7} C_VEL
LIN {X 0,Y 321.165,Z 367.724,A -85,B 0,C 180,E1 -15195.099,E2 -15195.099} C_VEL
LIN {X 0,Y 320.173,Z 375.629,A -85,B 0,C 180,E1 -15196.673,E2 -15196.673} C_VEL
LIN {X 0,Y 319.177,Z 383.328,A -85,B 0,C 180,E1 -15198.569,E2 -15198.569} C_VEL
LIN {X 0,Y 318.547,Z 389.513,A -85,B 0,C 180,E1 -15200.474,E2 -15200.474} C_VEL
LIN {X 0,Y 318.087,Z 394.401,A -85,B 0,C 180,E1 -15202.381,E2 -15202.381} C_VEL
LIN {X 0,Y 317.879,Z 398.022,A -85,B 0,C 180,E1 -15204.22,E2 -15204.22} C_VEL
LIN {X 0,Y 317.774,Z 400.834,A -85,B 0,C 180,E1 -15206.194,E2 -15206.194} C_VEL
LIN {X 0,Y 317.73,Z 402.097,A -85,B 0,C 180,E1 -15207.463,E2 -15207.463} C_VEL
LIN {X 0,Y 317.693,Z 402.946,A -85,B 0,C 180,E1 -15208.731,E2 -15208.731} C_VEL
LIN {X 0,Y 317.718,Z 403.351,A -85,B 0,C 180,E1 -15209.999,E2 -15209.999} C_VEL
LIN {X 0,Y 317.692,Z 403.361,A -85,B 0,C 180,E1 -15211.266,E2 -15211.266} C_VEL
LIN {X 0,Y 317.731,Z 402.981,A -85,B 0,C 180,E1 -15212.534,E2 -15212.534} C_VEL
LIN {X 0,Y 317.789,Z 402.2,A -85,B 0,C 180,E1 -15213.803,E2 -15213.803} C_VEL
LIN {X 0,Y 317.901,Z 400.086,A -85,B 0,C 180,E1 -15215.82,E2 -15215.82} C_VEL
LIN {X 0,Y 318.327,Z 396.06,A -85,B 0,C 180,E1 -15218.249,E2 -15218.249} C_VEL
LIN {X 0,Y 318.9,Z 391.713,A -85,B 0,C 180,E1 -15220.153,E2 -15220.153} C_VEL
LIN {X 0,Y 319.732,Z 386.186,A -85,B 0,C 180,E1 -15222.052,E2 -15222.052} C_VEL
LIN {X 0,Y 320.928,Z 379.299,A -85,B 0,C 180,E1 -15223.937,E2 -15223.937} C_VEL
LIN {X 0,Y 322.439,Z 370.716,A -85,B 0,C 180,E1 -15225.809,E2 -15225.809} C_VEL
LIN {X 0,Y 323.682,Z 362.206,A -85,B 0,C 180,E1 -15227.323,E2 -15227.323} C_VEL
LIN {X 0,Y 325.198,Z 352.317,A -85,B 0,C 180,E1 -15228.75,E2 -15228.75} C_VEL
LIN {X 0,Y 326.636,Z 341.846,A -85,B 0,C 180,E1 -15229.971,E2 -15229.971} C_VEL
LIN {X 0,Y 328.18,Z 330.3,A -85,B 0,C 180,E1 -15231.019,E2 -15231.019} C_VEL
LIN {X 0,Y 329.511,Z 317.157,A -85,B 0,C 180,E1 -15231.914,E2 -15231.914} C_VEL
LIN {X 0,Y 330.56,Z 304.005,A -85,B 0,C 180,E1 -15232.537,E2 -15232.537} C_VEL
LIN {X 0,Y 331.097,Z 289.461,A -85,B 0,C 180,E1 -15232.958,E2 -15232.958} C_VEL
LIN {X 0,Y 332.821,Z 228.967,A -85,B 0,C 180,E1 -15234.377,E2 -15234.377} C_VEL
LIN {X 0,Y 329.215,Z 208.262,A -85,B 0,C 180,E1 -15235.273,E2 -15235.273} C_VEL
LIN {X 0,Y 326.594,Z 196.78,A -85,B 0,C 180,E1 -15235.85,E2 -15235.85} C_VEL
LIN {X 0,Y 324.218,Z 190.848,A -85,B 0,C 180,E1 -15236.316,E2 -15236.316} C_VEL
LIN {X 0,Y 322.039,Z 180.424,A -85,B 0,C 180,E1 -15239.579,E2 -15239.579} C_VEL
LIN {X 0,Y 319.63,Z 170.525,A -85,B 0,C 180,E1 -15242.968,E2 -15242.968} C_VEL
LIN {X 0,Y 319.573,Z 170.172,A -85,B 0,C 180,E1 -15243.351,E2 -15243.351} C_VEL
LIN {X 0,Y 319.55,Z 170.181,A -85,B 0,C 180,E1 -15246.426,E2 -15246.426} C_VEL
LIN {X 0,Y 319.523,Z 170.183,A -85,B 0,C 180,E1 -15249.66,E2 -15249.66} C_VEL
LIN {X 0,Y 319.512,Z 170.186,A -85,B 0,C 180,E1 -15253.458,E2 -15253.458} C_VEL
LIN {X 0,Y 319.543,Z 170.179,A -85,B 0,C 180,E1 -15257.014,E2 -15257.014} C_VEL
LIN {X 0,Y 319.538,Z 170.181,A -85,B 0,C 180,E1 -15260.369,E2 -15260.369} C_VEL
LIN {X 0,Y 319.57,Z 170.178,A -85,B 0,C 180,E1 -15264.456,E2 -15264.456} C_VEL
LIN {X 0,Y 319.514,Z 170.182,A -85,B 0,C 180,E1 -15268.136,E2 -15268.136} C_VEL
LIN {X 0,Y 319.559,Z 170.176,A -85,B 0,C 180,E1 -15271.603,E2 -15271.603} C_VEL
LIN {X 0,Y 319.562,Z 170.177,A -85,B 0,C 180,E1 -15275.3,E2 -15275.3} C_VEL
LIN {X 0,Y 319.555,Z 170.176,A -85,B 0,C 180,E1 -15278.044,E2 -15278.044} C_VEL
LIN {X 0,Y 319.603,Z 170.17,A -85,B 0,C 180,E1 -15282.069,E2 -15282.069} C_VEL
LIN {X 0,Y 319.721,Z 170.155,A -85,B 0,C 180,E1 -15286.007,E2 -15286.007} C_VEL
LIN {X 0,Y 319.723,Z 170.155,A -85,B 0,C 180,E1 -15289.871,E2 -15289.871} C_VEL
LIN {X 0,Y 319.898,Z 170.133,A -85,B 0,C 180,E1 -15293.693,E2 -15293.693} C_VEL
LIN {X 0,Y 319.948,Z 170.128,A -85,B 0,C 180,E1 -15297.482,E2 -15297.482} C_VEL
LIN {X 0,Y 320.002,Z 170.124,A -85,B 0,C 180,E1 -15301.258,E2 -15301.258} C_VEL
LIN {X 0,Y 319.901,Z 170.133,A -85,B 0,C 180,E1 -15306.306,E2 -15306.306} C_VEL
LIN {X 0,Y 319.721,Z 170.159,A -85,B 0,C 180,E1 -15310.128,E2 -15310.128} C_VEL
LIN {X 0,Y 319.719,Z 170.157,A -85,B 0,C 180,E1 -15313.992,E2 -15313.992} C_VEL
LIN {X 0,Y 319.601,Z 170.174,A -85,B 0,C 180,E1 -15317.93,E2 -15317.93} C_VEL
LIN {X 0,Y 319.552,Z 170.181,A -85,B 0,C 180,E1 -15321.955,E2 -15321.955} C_VEL
LIN {X 0,Y 319.584,Z 170.426,A -85,B 0,C 180,E1 -15323.403,E2 -15323.403} C_VEL
LIN {X 0,Y 321.674,Z 179.002,A -85,B 0,C 180,E1 -15326.396,E2 -15326.396} C_VEL
LIN {X 0,Y 322.553,Z 182.851,A -85,B 0,C 180,E1 -15327.581,E2 -15327.581} C_VEL
LIN {X 0,Y 328.542,Z 196.178,A -85,B 0,C 180,E1 -15328.61,E2 -15328.61} C_VEL
LIN {X 0,Y 330.391,Z 201.36,A -85,B 0,C 180,E1 -15328.932,E2 -15328.932} C_VEL
LIN {X 0,Y 333.177,Z 215.861,A -85,B 0,C 180,E1 -15329.585,E2 -15329.585} C_VEL
LIN {X 0,Y 330.91,Z 290.981,A -85,B 0,C 180,E1 -15331.38,E2 -15331.38} C_VEL
LIN {X 0,Y 330.071,Z 304.136,A -85,B 0,C 180,E1 -15331.931,E2 -15331.931} C_VEL
LIN {X 0,Y 328.99,Z 317.163,A -85,B 0,C 180,E1 -15332.743,E2 -15332.743} C_VEL
LIN {X 0,Y 327.549,Z 329.662,A -85,B 0,C 180,E1 -15333.807,E2 -15333.807} C_VEL
LIN {X 0,Y 326.081,Z 340.69,A -85,B 0,C 180,E1 -15335.018,E2 -15335.018} C_VEL
LIN {X 0,Y 324.49,Z 350.921,A -85,B 0,C 180,E1 -15336.428,E2 -15336.428} C_VEL
LIN {X 0,Y 322.891,Z 360.833,A -85,B 0,C 180,E1 -15338.148,E2 -15338.148} C_VEL
LIN {X 0,Y 321.383,Z 369.649,A -85,B 0,C 180,E1 -15340.062,E2 -15340.062} C_VEL
LIN {X 0,Y 320.09,Z 376.93,A -85,B 0,C 180,E1 -15342.077,E2 -15342.077} C_VEL
LIN {X 0,Y 319.148,Z 382.899,A -85,B 0,C 180,E1 -15344.194,E2 -15344.194} C_VEL
LIN {X 0,Y 318.566,Z 386.79,A -85,B 0,C 180,E1 -15345.982,E2 -15345.982} C_VEL
LIN {X 0,Y 317.964,Z 390.676,A -85,B 0,C 180,E1 -15348.466,E2 -15348.466} C_VEL
LIN {X 0,Y 317.581,Z 392.784,A -85,B 0,C 180,E1 -15350.763,E2 -15350.763} C_VEL
LIN {X 0,Y 317.444,Z 393.6,A -85,B 0,C 180,E1 -15353.293,E2 -15353.293} C_VEL
LIN {X 0,Y 317.436,Z 393.205,A -85,B 0,C 180,E1 -15355.001,E2 -15355.001} C_VEL
LIN {X 0,Y 317.572,Z 391.616,A -85,B 0,C 180,E1 -15357.24,E2 -15357.24} C_VEL
LIN {X 0,Y 317.919,Z 388.566,A -85,B 0,C 180,E1 -15359.557,E2 -15359.557} C_VEL
LIN {X 0,Y 318.283,Z 384.814,A -85,B 0,C 180,E1 -15361.515,E2 -15361.515} C_VEL
LIN {X 0,Y 318.951,Z 378.755,A -85,B 0,C 180,E1 -15363.854,E2 -15363.854} C_VEL
LIN {X 0,Y 319.627,Z 372.74,A -85,B 0,C 180,E1 -15365.654,E2 -15365.654} C_VEL
LIN {X 0,Y 320.547,Z 365.048,A -85,B 0,C 180,E1 -15367.504,E2 -15367.504} C_VEL
LIN {X 0,Y 321.774,Z 355.253,A -85,B 0,C 180,E1 -15369.38,E2 -15369.38} C_VEL
LIN {X 0,Y 322.999,Z 344.965,A -85,B 0,C 180,E1 -15370.953,E2 -15370.953} C_VEL
LIN {X 0,Y 324.316,Z 333.431,A -85,B 0,C 180,E1 -15372.341,E2 -15372.341} C_VEL
LIN {X 0,Y 325.433,Z 321.668,A -85,B 0,C 180,E1 -15373.455,E2 -15373.455} C_VEL
LIN {X 0,Y 326.318,Z 309.845,A -85,B 0,C 180,E1 -15374.304,E2 -15374.304} C_VEL
LIN {X 0,Y 327.161,Z 296.484,A -85,B 0,C 180,E1 -15374.983,E2 -15374.983} C_VEL
LIN {X 0,Y 327.659,Z 282.77,A -85,B 0,C 180,E1 -15375.416,E2 -15375.416} C_VEL
LIN {X 0,Y 329.189,Z 213.673,A -85,B 0,C 180,E1 -15377.015,E2 -15377.015} C_VEL
LIN {X 0,Y 324.971,Z 190.829,A -85,B 0,C 180,E1 -15377.861,E2 -15377.861} C_VEL
LIN {X 0,Y 322.163,Z 182.633,A -85,B 0,C 180,E1 -15378.284,E2 -15378.284} C_VEL
LIN {X 0,Y 320.167,Z 171.796,A -85,B 0,C 180,E1 -15381.63,E2 -15381.63} C_VEL
LIN {X 0,Y 319.915,Z 170.16,A -85,B 0,C 180,E1 -15382.252,E2 -15382.252} C_VEL
LIN {X 0,Y 319.941,Z 170.133,A -85,B 0,C 180,E1 -15383.696,E2 -15383.696} C_VEL
LIN {X 0,Y 319.987,Z 170.126,A -85,B 0,C 180,E1 -15387.484,E2 -15387.484} C_VEL
LIN {X 0,Y 320.146,Z 170.106,A -85,B 0,C 180,E1 -15390.001,E2 -15390.001} C_VEL
LIN {X 0,Y 319.987,Z 170.124,A -85,B 0,C 180,E1 -15392.519,E2 -15392.519} C_VEL
LIN {X 0,Y 319.934,Z 170.13,A -85,B 0,C 180,E1 -15396.307,E2 -15396.307} C_VEL
LIN {X 0,Y 319.734,Z 170.156,A -85,B 0,C 180,E1 -15400.129,E2 -15400.129} C_VEL
LIN {X 0,Y 319.731,Z 170.156,A -85,B 0,C 180,E1 -15403.993,E2 -15403.993} C_VEL
LIN {X 0,Y 319.657,Z 170.163,A -85,B 0,C 180,E1 -15407.928,E2 -15407.928} C_VEL
LIN {X 0,Y 319.615,Z 170.169,A -85,B 0,C 180,E1 -15410.6,E2 -15410.6} C_VEL
LIN {X 0,Y 319.57,Z 170.179,A -85,B 0,C 180,E1 -15413.32,E2 -15413.32} C_VEL
LIN {X 0,Y 319.618,Z 170.165,A -85,B 0,C 180,E1 -15416.091,E2 -15416.091} C_VEL
LIN {X 0,Y 319.58,Z 170.176,A -85,B 0,C 180,E1 -15418.936,E2 -15418.936} C_VEL
LIN {X 0,Y 319.53,Z 170.18,A -85,B 0,C 180,E1 -15421.863,E2 -15421.863} C_VEL
LIN {X 0,Y 319.579,Z 170.17,A -85,B 0,C 180,E1 -15425.544,E2 -15425.544} C_VEL
LIN {X 0,Y 319.555,Z 170.176,A -85,B 0,C 180,E1 -15429.709,E2 -15429.709} C_VEL
LIN {X 0,Y 318.819,Z 170.272,A -85,B 0,C 180,E1 -15430.759,E2 -15430.759} C_VEL
LIN {X 0,Y 315.925,Z 170.632,A -85,B 0,C 180,E1 -15432.469,E2 -15432.469} C_VEL
LIN {X 0,Y 313.524,Z 170.927,A -85,B 0,C 180,E1 -15433.855,E2 -15433.855} C_VEL
LIN {X 0,Y 312.518,Z 171.054,A -85,B 0,C 180,E1 -15434.929,E2 -15434.929} C_VEL
LIN {X 0,Y 312.447,Z 171.057,A -85,B 0,C 180,E1 -15435.292,E2 -15435.292} C_VEL
LIN {X 0,Y 312.484,Z 171.05,A -85,B 0,C 180,E1 -15437.92,E2 -15437.92} C_VEL
LIN {X 0,Y 312.495,Z 171.056,A -85,B 0,C 180,E1 -15440.971,E2 -15440.971} C_VEL
LIN {X 0,Y 312.532,Z 171.054,A -85,B 0,C 180,E1 -15444.221,E2 -15444.221} C_VEL
LIN {X 0,Y 312.502,Z 171.055,A -85,B 0,C 180,E1 -15447.334,E2 -15447.334} C_VEL
LIN {X 0,Y 312.508,Z 171.055,A -85,B 0,C 180,E1 -15451.292,E2 -15451.292} C_VEL
LIN {X 0,Y 312.55,Z 171.051,A -85,B 0,C 180,E1 -15454.709,E2 -15454.709} C_VEL
LIN {X 0,Y 312.566,Z 171.045,A -85,B 0,C 180,E1 -15457.528,E2 -15457.528} C_VEL
LIN {X 0,Y 312.64,Z 171.039,A -85,B 0,C 180,E1 -15461.657,E2 -15461.657} C_VEL
LIN {X 0,Y 312.696,Z 171.031,A -85,B 0,C 180,E1 -15465.687,E2 -15465.687} C_VEL
LIN {X 0,Y 312.687,Z 171.034,A -85,B 0,C 180,E1 -15469.642,E2 -15469.642} C_VEL
LIN {X 0,Y 312.798,Z 171.019,A -85,B 0,C 180,E1 -15472.253,E2 -15472.253} C_VEL
LIN {X 0,Y 312.689,Z 171.032,A -85,B 0,C 180,E1 -15474.843,E2 -15474.843} C_VEL
LIN {X 0,Y 312.981,Z 170.994,A -85,B 0,C 180,E1 -15478.714,E2 -15478.714} C_VEL
LIN {X 0,Y 312.91,Z 170.996,A -85,B 0,C 180,E1 -15482.575,E2 -15482.575} C_VEL
LIN {X 0,Y 312.84,Z 171.011,A -85,B 0,C 180,E1 -15486.45,E2 -15486.45} C_VEL
LIN {X 0,Y 312.754,Z 171.025,A -85,B 0,C 180,E1 -15489.051,E2 -15489.051} C_VEL
LIN {X 0,Y 312.635,Z 171.039,A -85,B 0,C 180,E1 -15492.992,E2 -15492.992} C_VEL
LIN {X 0,Y 312.623,Z 171.037,A -85,B 0,C 180,E1 -15495.651,E2 -15495.651} C_VEL
LIN {X 0,Y 312.538,Z 171.053,A -85,B 0,C 180,E1 -15499.713,E2 -15499.713} C_VEL
LIN {X 0,Y 312.517,Z 171.055,A -85,B 0,C 180,E1 -15502.775,E2 -15502.775} C_VEL
LIN {X 0,Y 312.485,Z 171.054,A -85,B 0,C 180,E1 -15506.732,E2 -15506.732} C_VEL
LIN {X 0,Y 312.496,Z 171.058,A -85,B 0,C 180,E1 -15509.656,E2 -15509.656} C_VEL
LIN {X 0,Y 312.523,Z 171.05,A -85,B 0,C 180,E1 -15513.689,E2 -15513.689} C_VEL
LIN {X 0,Y 312.516,Z 171.056,A -85,B 0,C 180,E1 -15517.387,E2 -15517.387} C_VEL
LIN {X 0,Y 312.444,Z 171.064,A -85,B 0,C 180,E1 -15520.717,E2 -15520.717} C_VEL
LIN {X 0,Y 312.453,Z 171.062,A -85,B 0,C 180,E1 -15524.21,E2 -15524.21} C_VEL
LIN {X 0,Y 312.457,Z 171.062,A -85,B 0,C 180,E1 -15527.925,E2 -15527.925} C_VEL
LIN {X 0,Y 312.478,Z 171.06,A -85,B 0,C 180,E1 -15531.925,E2 -15531.925} C_VEL
LIN {X 0,Y 312.531,Z 171.055,A -85,B 0,C 180,E1 -15534.219,E2 -15534.219} C_VEL
LIN {X 0,Y 312.502,Z 171.058,A -85,B 0,C 180,E1 -15537.333,E2 -15537.333} C_VEL
LIN {X 0,Y 312.523,Z 171.215,A -85,B 0,C 180,E1 -15539.041,E2 -15539.041} C_VEL
LIN {X 0,Y 314.673,Z 181.562,A -85,B 0,C 180,E1 -15542.337,E2 -15542.337} C_VEL
LIN {X 0,Y 316.445,Z 191.408,A -85,B 0,C 180,E1 -15545.274,E2 -15545.274} C_VEL
LIN {X 0,Y 316.688,Z 193.11,A -85,B 0,C 180,E1 -15545.424,E2 -15545.424} C_VEL
LIN {X 0,Y 322.36,Z 228.727,A -85,B 0,C 180,E1 -15546.722,E2 -15546.722} C_VEL
LIN {X 0,Y 320.669,Z 299.521,A -85,B 0,C 180,E1 -15548.42,E2 -15548.42} C_VEL
LIN {X 0,Y 319.852,Z 313.261,A -85,B 0,C 180,E1 -15548.995,E2 -15548.995} C_VEL
LIN {X 0,Y 318.889,Z 325.739,A -85,B 0,C 180,E1 -15549.772,E2 -15549.772} C_VEL
LIN {X 0,Y 317.694,Z 337.709,A -85,B 0,C 180,E1 -15550.787,E2 -15550.787} C_VEL
LIN {X 0,Y 316.429,Z 349.213,A -85,B 0,C 180,E1 -15552.05,E2 -15552.05} C_VEL
LIN {X 0,Y 315.203,Z 359.642,A -85,B 0,C 180,E1 -15553.49,E2 -15553.49} C_VEL
LIN {X 0,Y 314.034,Z 368.909,A -85,B 0,C 180,E1 -15555.085,E2 -15555.085} C_VEL
LIN {X 0,Y 312.851,Z 377.955,A -85,B 0,C 180,E1 -15557.017,E2 -15557.017} C_VEL
LIN {X 0,Y 311.975,Z 385.223,A -85,B 0,C 180,E1 -15558.959,E2 -15558.959} C_VEL
LIN {X 0,Y 311.349,Z 390.997,A -85,B 0,C 180,E1 -15560.907,E2 -15560.907} C_VEL
LIN {X 0,Y 310.931,Z 395.527,A -85,B 0,C 180,E1 -15562.857,E2 -15562.857} C_VEL
LIN {X 0,Y 310.716,Z 398.949,A -85,B 0,C 180,E1 -15564.808,E2 -15564.808} C_VEL
LIN {X 0,Y 310.688,Z 400.643,A -85,B 0,C 180,E1 -15566.107,E2 -15566.107} C_VEL
LIN {X 0,Y 310.654,Z 401.925,A -85,B 0,C 180,E1 -15567.405,E2 -15567.405} C_VEL
LIN {X 0,Y 310.61,Z 402.801,A -85,B 0,C 180,E1 -15568.702,E2 -15568.702} C_VEL
LIN {X 0,Y 310.631,Z 403.232,A -85,B 0,C 180,E1 -15569.999,E2 -15569.999} C_VEL
LIN {X 0,Y 310.609,Z 403.258,A -85,B 0,C 180,E1 -15571.295,E2 -15571.295} C_VEL
LIN {X 0,Y 310.656,Z 402.895,A -85,B 0,C 180,E1 -15572.592,E2 -15572.592} C_VEL
LIN {X 0,Y 310.705,Z 402.138,A -85,B 0,C 180,E1 -15573.89,E2 -15573.89} C_VEL
LIN {X 0,Y 310.815,Z 400.261,A -85,B 0,C 180,E1 -15575.78,E2 -15575.78} C_VEL
LIN {X 0,Y 311.119,Z 397.289,A -85,B 0,C 180,E1 -15577.788,E2 -15577.788} C_VEL
LIN {X 0,Y 311.674,Z 393.356,A -85,B 0,C 180,E1 -15579.735,E2 -15579.735} C_VEL
LIN {X 0,Y 312.491,Z 388.293,A -85,B 0,C 180,E1 -15581.676,E2 -15581.676} C_VEL
LIN {X 0,Y 313.537,Z 381.947,A -85,B 0,C 180,E1 -15583.611,E2 -15583.611} C_VEL
LIN {X 0,Y 315.112,Z 374.007,A -85,B 0,C 180,E1 -15585.522,E2 -15585.522} C_VEL
LIN {X 0,Y 316.404,Z 365.338,A -85,B 0,C 180,E1 -15587.229,E2 -15587.229} C_VEL
LIN {X 0,Y 318.125,Z 355.063,A -85,B 0,C 180,E1 -15588.848,E2 -15588.848} C_VEL
LIN {X 0,Y 319.829,Z 343.794,A -85,B 0,C 180,E1 -15590.247,E2 -15590.247} C_VEL
LIN {X 0,Y 321.404,Z 332.805,A -85,B 0,C 180,E1 -15591.315,E2 -15591.315} C_VEL
LIN {X 0,Y 322.757,Z 320.745,A -85,B 0,C 180,E1 -15592.229,E2 -15592.229} C_VEL
LIN {X 0,Y 323.913,Z 307.392,A -85,B 0,C 180,E1 -15592.945,E2 -15592.945} C_VEL
LIN {X 0,Y 324.623,Z 293.497,A -85,B 0,C 180,E1 -15593.421,E2 -15593.421} C_VEL
LIN {X 0,Y 326.527,Z 229.847,A -85,B 0,C 180,E1 -15594.95,E2 -15594.95} C_VEL
LIN {X 0,Y 323.279,Z 210.795,A -85,B 0,C 180,E1 -15595.794,E2 -15595.794} C_VEL
LIN {X 0,Y 320.748,Z 199.571,A -85,B 0,C 180,E1 -15596.376,E2 -15596.376} C_VEL
LIN {X 0,Y 317.069,Z 190.809,A -85,B 0,C 180,E1 -15597.068,E2 -15597.068} C_VEL
LIN {X 0,Y 314.766,Z 180.164,A -85,B 0,C 180,E1 -15600.531,E2 -15600.531} C_VEL
LIN {X 0,Y 312.52,Z 171.162,A -85,B 0,C 180,E1 -15603.809,E2 -15603.809} C_VEL
LIN {X 0,Y 312.505,Z 171.061,A -85,B 0,C 180,E1 -15607.386,E2 -15607.386} C_VEL
LIN {X 0,Y 312.435,Z 171.067,A -85,B 0,C 180,E1 -15610.715,E2 -15610.715} C_VEL
LIN {X 0,Y 312.443,Z 171.063,A -85,B 0,C 180,E1 -15614.208,E2 -15614.208} C_VEL
LIN {X 0,Y 312.447,Z 171.067,A -85,B 0,C 180,E1 -15617.923,E2 -15617.923} C_VEL
LIN {X 0,Y 312.475,Z 171.057,A -85,B 0,C 180,E1 -15621.921,E2 -15621.921} C_VEL
LIN {X 0,Y 312.521,Z 171.056,A -85,B 0,C 180,E1 -15624.218,E2 -15624.218} C_VEL
LIN {X 0,Y 312.492,Z 171.061,A -85,B 0,C 180,E1 -15627.332,E2 -15627.332} C_VEL
LIN {X 0,Y 312.495,Z 171.059,A -85,B 0,C 180,E1 -15631.291,E2 -15631.291} C_VEL
LIN {X 0,Y 312.536,Z 171.055,A -85,B 0,C 180,E1 -15634.706,E2 -15634.706} C_VEL
LIN {X 0,Y 312.513,Z 171.058,A -85,B 0,C 180,E1 -15638.91,E2 -15638.91} C_VEL
LIN {X 0,Y 312.567,Z 171.049,A -85,B 0,C 180,E1 -15643.004,E2 -15643.004} C_VEL
LIN {X 0,Y 312.674,Z 171.032,A -85,B 0,C 180,E1 -15645.685,E2 -15645.685} C_VEL
LIN {X 0,Y 312.673,Z 171.032,A -85,B 0,C 180,E1 -15649.64,E2 -15649.64} C_VEL
LIN {X 0,Y 312.807,Z 171.014,A -85,B 0,C 180,E1 -15652.252,E2 -15652.252} C_VEL
LIN {X 0,Y 312.686,Z 171.036,A -85,B 0,C 180,E1 -15654.841,E2 -15654.841} C_VEL
LIN {X 0,Y 312.955,Z 171.001,A -85,B 0,C 180,E1 -15658.713,E2 -15658.713} C_VEL
LIN {X 0,Y 312.969,Z 171,A -85,B 0,C 180,E1 -15661.286,E2 -15661.286} C_VEL
LIN {X 0,Y 312.845,Z 171.012,A -85,B 0,C 180,E1 -15666.449,E2 -15666.449} C_VEL
LIN {X 0,Y 312.738,Z 171.025,A -85,B 0,C 180,E1 -15669.05,E2 -15669.05} C_VEL
LIN {X 0,Y 312.62,Z 171.044,A -85,B 0,C 180,E1 -15672.991,E2 -15672.991} C_VEL
LIN {X 0,Y 312.609,Z 171.044,A -85,B 0,C 180,E1 -15675.651,E2 -15675.651} C_VEL
LIN {X 0,Y 312.525,Z 171.056,A -85,B 0,C 180,E1 -15679.713,E2 -15679.713} C_VEL
LIN {X 0,Y 312.531,Z 171.173,A -85,B 0,C 180,E1 -15682.627,E2 -15682.627} C_VEL
LIN {X 0,Y 314.217,Z 177.952,A -85,B 0,C 180,E1 -15685.148,E2 -15685.148} C_VEL
LIN {X 0,Y 315.379,Z 182.897,A -85,B 0,C 180,E1 -15686.792,E2 -15686.792} C_VEL
LIN {X 0,Y 322.208,Z 197.906,A -85,B 0,C 180,E1 -15688.01,E2 -15688.01} C_VEL
LIN {X 0,Y 324.469,Z 203.93,A -85,B 0,C 180,E1 -15688.414,E2 -15688.414} C_VEL
LIN {X 0,Y 326.973,Z 217.429,A -85,B 0,C 180,E1 -15689.031,E2 -15689.031} C_VEL
LIN {X 0,Y 324.567,Z 291.172,A -85,B 0,C 180,E1 -15690.828,E2 -15690.828} C_VEL
LIN {X 0,Y 323.693,Z 304.209,A -85,B 0,C 180,E1 -15691.384,E2 -15691.384} C_VEL
LIN {X 0,Y 322.603,Z 316.931,A -85,B 0,C 180,E1 -15692.19,E2 -15692.19} C_VEL
LIN {X 0,Y 321.256,Z 328.293,A -85,B 0,C 180,E1 -15693.155,E2 -15693.155} C_VEL
LIN {X 0,Y 319.529,Z 340.626,A -85,B 0,C 180,E1 -15694.512,E2 -15694.512} C_VEL
LIN {X 0,Y 317.931,Z 350.531,A -85,B 0,C 180,E1 -15695.89,E2 -15695.89} C_VEL
LIN {X 0,Y 316.226,Z 360.559,A -85,B 0,C 180,E1 -15697.647,E2 -15697.647} C_VEL
LIN {X 0,Y 314.963,Z 367.617,A -85,B 0,C 180,E1 -15699.162,E2 -15699.162} C_VEL
LIN {X 0,Y 313.74,Z 374.272,A -85,B 0,C 180,E1 -15700.893,E2 -15700.893} C_VEL
